FUNCTION_BLOCK "Asse_611U"	// FB 16
TITLE = Axis 611U management
AUTHOR : Cellini
VERSION : 0.1
VAR_INPUT
  IO_LAddr : INT ;	//Logic address of the inputs/outputs
END_VAR
VAR
  In_Profibus : STRUCT 	//Inputs from 611U (via Profibus)
   PKW : STRUCT 	//Parameter area of the Profibus telegram
    PKE : WORD ;
    IND : WORD ;
    PWE : DINT ;
   END_STRUCT ;
   PZD : STRUCT 	//Process data area of the Profibus telegram
    ZSW1 : STRUCT 	//Status word 1
     Bit8 : BOOL ;	//Following error (0=following error outside the window error)
     Bit9 : BOOL ;	//DP control requested (1=DP master is requested to accept control)
     Bit10 : BOOL ;	//Reference position reached (1=end of traversing block reached)
     Bit11 : BOOL ;	//Reference point set (1=axis is referenced)
     Bit12 : BOOL ;	//Setpoint acknowledge (1=the traversing task is processed)
     Bit13 : BOOL ;	//Drive stationery (1=drive is not in movement)
     Bit14 : BOOL ;	//External block change selected
     Bit15 : BOOL ;	//Request passive referencing
     Bit0 : BOOL ;	//Ready to switch-on (1=ready to power-up)
     Bit1 : BOOL ;	//Ready or no fault (1=drive ready or no fault present)
     Bit2 : BOOL ;	//Controller enable (1=speed controller active and setpoint can be accepted)
     Bit3 : BOOL ;	//Fault present (1=fault present)
     Bit4 : BOOL ;	//No OFF2 (1=OFF2 not present)
     Bit5 : BOOL ;	//No OFF3 (1=OFF3 not present)
     Bit6 : BOOL ;	//Switch-on inhibit (1=power-on inhibit)
     Bit7 : BOOL ;	//Alarm present (1=alarm present)
    END_STRUCT ;
    AktSatz : STRUCT 	//Actual block status word
     Bit8 : BOOL ;	//Reserved
     Bit9 : BOOL ;	//Reserved
     Bit10 : BOOL ;	//Reserved
     Bit11 : BOOL ;	//Reserved
     Bit12 : BOOL ;	//Reserved
     Bit13 : BOOL ;	//Reserved
     Bit14 : BOOL ;	//Reserved
     Bit15 : BOOL ;	//MDI Active
     Bit0 : BOOL ;	//Bit 0 block selected
     Bit1 : BOOL ;	//Bit 1 block selected
     Bit2 : BOOL ;	//Bit 2 block selected
     Bit3 : BOOL ;	//Bit 3 block selected
     Bit4 : BOOL ;	//Bit 4 block selected
     Bit5 : BOOL ;	//Bit 5 block selected
     Bit6 : BOOL ;	//Reserved
     Bit7 : BOOL ;	//Reserved
    END_STRUCT ;
    PosZsw : STRUCT 	//Position status word
     Bit8 : BOOL ;	//Cam switching signal 1
     Bit9 : BOOL ;	//Cam switching signal 2
     Bit10 : BOOL ;	//Direct output 1 via the traversing block
     Bit11 : BOOL ;	//Direct output 2 via the traversing block
     Bit12 : BOOL ;	//Fixed endstop reached
     Bit13 : BOOL ;	//Fixed endstop clamping torque reached
     Bit14 : BOOL ;	//Traverse to fixed endstop active
     Bit15 : BOOL ;	//Teach-In executed
     Bit0 : BOOL ;	//Tracking mode active (1=tracking mode active)
     Bit1 : BOOL ;	//Velocity limiting (1=velocity is limited)
     Bit2 : BOOL ;	//Setpoint stationary (1=axis stationary on the setpoint side)
     Bit3 : BOOL ;	//In synchronism (1=slave drive is synchronized with the master drive)
     Bit4 : BOOL ;	//Axis moves forwards
     Bit5 : BOOL ;	//Axis moves backwards
     Bit6 : BOOL ;	//Minus software limit switch actuated
     Bit7 : BOOL ;	//Plus software limit switch actuated
    END_STRUCT ;
    ZSW2 : STRUCT 	//Status word 2
     Bit8 : BOOL ;	//Suppress fault 608 active
     Bit9 : BOOL ;	//n.u. (used only in the n-set mode)
     Bit10 : BOOL ;	//n.u. (used only in the n-set mode)
     Bit11 : BOOL ;	//n.u. (used only in the n-set mode)
     Bit12 : BOOL ;	//Slave sign-of-life
     Bit13 : BOOL ;	//Slave sign-of-life
     Bit14 : BOOL ;	//Slave sign-of-life
     Bit15 : BOOL ;	//Slave sign-of-life
     Bit0 : BOOL ;	//Bit 0 parameter set
     Bit1 : BOOL ;	//Bit 1 parameter set
     Bit2 : BOOL ;	//Bit 2 parameter set
     Bit3 : BOOL ;	//First speed setpoint filter inactive
     Bit4 : BOOL ;	//Rump-function generator inactive
     Bit5 : BOOL ;	//Open holding brake
     Bit6 : BOOL ;	//Integrator inhibit
     Bit7 : BOOL ;	//Parking axis selected
    END_STRUCT ;
    XretrP : DINT ;	//Actual position value
    DIG_IN : STRUCT 	//Digital inputs status
     Bit8 : BOOL ;
     Bit9 : BOOL ;
     Bit10 : BOOL ;
     Bit11 : BOOL ;
     Bit12 : BOOL ;
     Bit13 : BOOL ;
     Bit14 : BOOL ;
     Bit15 : BOOL ;
     Bit0 : BOOL ;	//Axis on home cam
     Bit1 : BOOL ;	//Axis on minus extra-corse limit switch
     Bit2 : BOOL ;	//Axis on plus extra-corse limit switch
     Bit3 : BOOL ;
     Bit4 : BOOL ;
     Bit5 : BOOL ;
     Bit6 : BOOL ;
     Bit7 : BOOL ;
    END_STRUCT ;
   END_STRUCT ;
  END_STRUCT ;
  Out_Profibus : STRUCT 	//Outputs to 611U (via Profibus)
   PKW : STRUCT 	//Parameter area of the Profibus telegram
    PKE : WORD ;
    IND : WORD ;
    PWE : DINT ;
   END_STRUCT ;
   PZD : STRUCT 	//Process data area of the Profibus telegram
    STW1 : STRUCT 	//Control word 1
     Bit8 : BOOL ;	//JOG1 (1=the drive traverse with the speed in P0108)
     Bit9 : BOOL ;	//JOG2 (1=the drive traverse with the speed in P0109)
     Bit10 : BOOL ;	//Control requested (Should be set 1 when ZSW1.9=1)
     Bit11 : BOOL ;	//Stop referencing (1=start the referencing point approach)
     Bit12 : BOOL ;	//Opening the holding brake for test purposes
     Bit13 : BOOL ;	//External block change (With a edge the external block changing is initiated)
     Bit14 : BOOL ;	//Reserved
     Bit15 : BOOL ;	//Request passive referencing
     Bit0 : BOOL ;	//OFF1 (1=enable)
     Bit1 : BOOL ;	//OFF2 (1=enable)
     Bit2 : BOOL ;	//OFF3 (1=enable)
     Bit3 : BOOL ;	//Pulse inhibit (0=the motor stop for inertia)
     Bit4 : BOOL ;	//Reject travel task (0=stop the motor and delete the distance to go)
     Bit5 : BOOL ;	//Intermediate stop (0=stop the motor but the process is continued with 0/1 edge)
     Bit6 : BOOL ;	//Activate travel task (With a edge the traversing block selected is started)
     Bit7 : BOOL ;	//Reset the fault memory (1=Reset the fault memory)
    END_STRUCT ;
    SatzAnw : STRUCT 	//Block selection control word
     Bit8 : BOOL ;	//Reserved
     Bit9 : BOOL ;	//Reserved
     Bit10 : BOOL ;	//Reserved
     Bit11 : BOOL ;	//Reserved
     Bit12 : BOOL ;	//Reserved
     Bit13 : BOOL ;	//Reserved
     Bit14 : BOOL ;	//Reserved
     Bit15 : BOOL ;	//Activate MDI
     Bit0 : BOOL ;	//Bit 0 block selection
     Bit1 : BOOL ;	//Bit 1 block selection
     Bit2 : BOOL ;	//Bit 2 block selection
     Bit3 : BOOL ;	//Bit 3 block selection
     Bit4 : BOOL ;	//Bit 4 block selection
     Bit5 : BOOL ;	//Bit 5 block selection
     Bit6 : BOOL ;	//Reserved
     Bit7 : BOOL ;	//Reserved
    END_STRUCT ;
    PosStw : STRUCT 	//Position control word
     Bit8 : BOOL ;	//Reserved
     Bit9 : BOOL ;	//Reserved
     Bit10 : BOOL ;	//Reserved
     Bit11 : BOOL ;	//Reserved
     Bit12 : BOOL ;	//Reserved
     Bit13 : BOOL ;	//Reserved
     Bit14 : BOOL ;	//Reserved
     Bit15 : BOOL ;	//Reserved
     Bit0 : BOOL ;	//Tracking operation (1=select tracking operation)
     Bit1 : BOOL ;	//Set reference point (0/1 edge=P0160 is assigned as actual value)
     Bit2 : BOOL ;	//Reference cams (1=the axis is located at reference cam)
     Bit3 : BOOL ;	//Fixed endstop (1=fixed endstop reached)
     Bit4 : BOOL ;	//Activate the coupling (0/1 edge=activate coupling set via P0410)
     BIt5 : BOOL ;	//Incremental jogging (1=jog in velocity and increments)
     Bit6 : BOOL ;	//Activate Teach-In (0/1=Activate Teach-In; 1/0=Reset Teach-In)
     Bit7 : BOOL ;	//Invert the angular encoder input
    END_STRUCT ;
    STW2 : STRUCT 	//Control word 2
     Bit8 : BOOL ;	//Suppress fault 608
     Bit9 : BOOL ;	//n.u. (used only in the n-set mode)
     Bit10 : BOOL ;	//n.u. (used only in the n-set mode)
     Bit11 : BOOL ;	//n.u. (used only in the n-set mode)
     Bit12 : BOOL ;	//Master sign-of-life
     Bit13 : BOOL ;	//Master sign-of-life
     Bit14 : BOOL ;	//Master sign-of-life
     Bit15 : BOOL ;	//Master sign-of-life
     Bit0 : BOOL ;	//Bit 0 parameter set changeover
     Bit1 : BOOL ;	//Bit 1 parameter set changeover
     Bit2 : BOOL ;	//Bit 2 parameter set changeover
     Bit3 : BOOL ;	//First speed setpoint filter disabled
     Bit4 : BOOL ;	//Rump-function generator enabled
     Bit5 : BOOL ;	//Reserved
     Bit6 : BOOL ;	//Integrator inhibit
     Bit7 : BOOL ;	//Select parking axis
    END_STRUCT ;
    Over : INT ;	//Percentage value for the velocity override
   END_STRUCT ;
  END_STRUCT ;
  Enable : BOOL ;	//Enable the drive
  Reset_Alarms : BOOL ;	//Reset the alarms
  Reset_Axis : BOOL ;	//Stop all the movements
  Start_Inc : BOOL ;	//Start incremental movement
  Start_Abs : BOOL ;	//Start absolute movement
  Start_Rep : BOOL ;	//Start repositioning movement
  Start_Ref : BOOL ;	//Start referencing movement
  Stop : BOOL ;	//Intermediate stop movement
  Jog_Forward : BOOL ;	//Jog forward command
  Jog_Backward : BOOL ;	//Jog backward command
  STAT58 : BOOL ;	//Reserved
  STAT57 : BOOL ;	//Reserved
  STAT56 : BOOL ;	//Reserved
  STAT55 : BOOL ;	//Reserved
  STAT54 : BOOL ;	//Reserved
  STAT53 : BOOL ;	//Reserved
  Step1_Inc : BOOL ;	//Step 1 for incremental movement management
  Step2_Inc : BOOL ;	//Step 2 for incremental movement management
  Step1_Abs : BOOL ;	//Step 1 for absolute movement management
  Step2_Abs : BOOL ;	//Step 2 for absolute movement management
  STAT36 : BOOL ;	//Reserved
  STAT35 : BOOL ;	//Reserved
  STAT34 : BOOL ;	//Reserved
  STAT33 : BOOL ;	//Reserved
  InZeroPosition : BOOL ;	//Axis in "zero" position
  AxisStationery : BOOL ;	//Axis stationery
  DriveOK : BOOL ;	//Drive OK
  BrakeOpen : BOOL ;	//Open holding brake request
  AxisOnHWHomeCam : BOOL ;	//Axis on hardware home cam
  AxisOnHWSwitchN : BOOL ;	//Axis on minus hardware extra-corse limit switch
  AxisOnHWSwitchP : BOOL ;	//Axis on plus hardware extra-corse limit switch
  AxisOnSWSwitchN : BOOL ;	//Axis on minus software extra-corse limit switch
  AxisOnSWSwitchP : BOOL ;	//Axis on plus software extra-corse limit switch
  STAT69 : BOOL ;	//Reserved
  STAT67 : BOOL ;	//Reserved
  STAT66 : BOOL ;	//Reserved
  STAT65 : BOOL ;	//Reserved
  STAT64 : BOOL ;	//Reserved
  STAT63 : BOOL ;	//Reserved
  STAT70 : BOOL ;	//Reserved
  Aux1 : BOOL ;	//Auxiliary for edge management
  Aux2 : BOOL ;	//Auxiliary for edge management
  Aux3 : BOOL ;	//Auxiliary for edge management
  Aux4 : BOOL ;	//Auxiliary for edge management
  Aux5 : BOOL ;	//Auxiliary for edge management
  Aux6 : BOOL ;	//Auxiliary for edge management
  Aux7 : BOOL ;	//Auxiliary for edge management
  Aux8 : BOOL ;	//Auxiliary for edge management
  Target_Inc : DINT ;	//Target for the incremental movement
  Target_Abs : DINT ;	//Target for the absolute movement
  DistanceToGo_Abs : DINT ;	//Difference between actual and new position
  Override : INT ;	//Percentage value for the velocity override
  ActualPosition : DINT ;	//Actual position value
END_VAR
VAR_TEMP
  tempAR1 : DWORD ;
  tempAR2 : DWORD ;
  tempSRC : ANY ;
  tempDST : ANY ;
  tempDWORD_1 : DWORD ;
  tempWORD_1 : WORD ;
  tempINT : INT ;
  tempDWORD_2 : DWORD ;
END_VAR
BEGIN
NETWORK
TITLE = Mapping of the inputs
      L     #IO_LAddr;
      SLD   3;
      T     #tempDWORD_1;
      L     P##In_Profibus;
      T     #tempDWORD_2;
      L     11;
NXT1: T     #tempINT;
      L     PIW [#tempDWORD_1];
      T     DIW [#tempDWORD_2];
      L     #tempDWORD_1;
      L     P#2.0;
      +D;
      T     #tempDWORD_1;
      L     #tempDWORD_2;
      L     P#2.0;
      +D;
      T     #tempDWORD_2;
      L     #tempINT;
      LOOP  NXT1;
NETWORK
TITLE = Status
//Axis stationery
      A     #In_Profibus.PZD.ZSW1.Bit13;
      AN    #In_Profibus.PZD.ZSW1.Bit12;
      =     #AxisStationery;
//Drive OK
      A     #In_Profibus.PZD.ZSW1.Bit0;
      A     #In_Profibus.PZD.ZSW1.Bit1;
      A     #In_Profibus.PZD.ZSW1.Bit2;
      AN    #In_Profibus.PZD.ZSW1.Bit3;
      A     #In_Profibus.PZD.ZSW1.Bit4;
      A     #In_Profibus.PZD.ZSW1.Bit5;
      A     #In_Profibus.PZD.ZSW1.Bit8;
      =     #DriveOK;
//Open holding brake request
      A     #In_Profibus.PZD.ZSW2.Bit5;
      =     #BrakeOpen;
//Axis on hardware home cam
      A     #In_Profibus.PZD.DIG_IN.Bit0;
      =     #AxisOnHWHomeCam;
//Axis on hardware minus extra-course limit switch
      A     #In_Profibus.PZD.DIG_IN.Bit1;
      =     #AxisOnHWSwitchN;
//Axis on hardware plus extra-course limit switch
      A     #In_Profibus.PZD.DIG_IN.Bit2;
      =     #AxisOnHWSwitchP;
//Axis on software minus extra-course limit switch
      A     #In_Profibus.PZD.PosZsw.Bit6;
      =     #AxisOnSWSwitchN;
//Axis on software plus extra-course limit switch
      A     #In_Profibus.PZD.PosZsw.Bit7;
      =     #AxisOnSWSwitchP;
//Actual position value
      L     #In_Profibus.PZD.XretrP;
      T     #ActualPosition;
NETWORK
TITLE = Commands
//Enable the drive
      A     #Enable;
      =     #Out_Profibus.PZD.STW1.Bit0;
      =     #Out_Profibus.PZD.STW1.Bit1;
      =     #Out_Profibus.PZD.STW1.Bit2;
      A     "On";
      =     #Out_Profibus.PZD.STW1.Bit3;
//Erase all the movements
      O     #Reset_Axis;
      O     #In_Profibus.PZD.ZSW1.Bit3;
      ON    #In_Profibus.PZD.ZSW1.Bit8;
      R     #Start_Inc;
      R     #Step1_Inc;
      R     #Step2_Inc;
      R     #Start_Abs;
      R     #Step1_Abs;
      R     #Step2_Abs;
      R     #Start_Rep;
      R     #Start_Ref;
      R     #Out_Profibus.PZD.STW1.Bit11;
      R     #Out_Profibus.PZD.STW1.Bit6;
//Stop the axis and erase the distance to go
      AN    #Reset_Axis;
      =     #Out_Profibus.PZD.STW1.Bit4;
//Intermediate stop the axis (the movement continued with a 0/1 edge)
      AN    #Stop;
      =     #Out_Profibus.PZD.STW1.Bit5;
//Reset alarms
      A     #Reset_Alarms;
      =     #Out_Profibus.PZD.STW1.Bit7;
//Control request (611U<->PLC communication)
      A     #In_Profibus.PZD.ZSW1.Bit9;
      =     #Out_Profibus.PZD.STW1.Bit10;
//Velocity override
      L     #Override;
      T     #Out_Profibus.PZD.Over;
NETWORK
TITLE = Movement in incremental mode
//Reset the incremental movement if the axis is the distance to go is minus then 0,05mm
      A     #Start_Inc;
      A(;
      L     #Target_Inc;
      L     50;
      <D;
      );
      A(;
      L     #Target_Inc;
      L     -50;
      >D;
      );
      R     #Start_Inc;
//Select the travel block (Block number 2=000010)
      A     #Start_Inc;
      R     #Out_Profibus.PZD.SatzAnw.Bit0;
      S     #Out_Profibus.PZD.SatzAnw.Bit1;
      R     #Out_Profibus.PZD.SatzAnw.Bit2;
      R     #Out_Profibus.PZD.SatzAnw.Bit3;
      R     #Out_Profibus.PZD.SatzAnw.Bit4;
      R     #Out_Profibus.PZD.SatzAnw.Bit5;
//Load the new position of the travel block
      A     #Start_Inc;
      AN    #Step1_Inc;
      AN    #Step2_Inc;
      S     #Step1_Inc;
      JCN   L001;
      L     #Target_Inc;
      T     #Out_Profibus.PKW.PWE;
      L     W#16#8051;
      T     #Out_Profibus.PKW.PKE;
      L     2;
      T     #Out_Profibus.PKW.IND;
L001: NOP   0;
//Check if the 611U received the change
      A     #Start_Inc;
      A     #Step1_Inc;
      AN    #Step2_Inc;
      A(;
      L     #Out_Profibus.PKW.PWE;
      L     #In_Profibus.PKW.PWE;
      ==D;
      );
      A(;
      L     W#16#5051;
      L     #In_Profibus.PKW.PKE;
      ==I;
      );
      A(;
      L     #Out_Profibus.PKW.IND;
      L     #In_Profibus.PKW.IND;
      ==I;
      );
      S     #Step2_Inc;
//Start travel task
      A     #Start_Inc;
      A     #Step1_Inc;
      A     #Step2_Inc;
      A(;
      L     #Target_Inc;
      L     #In_Profibus.PKW.PWE;
      ==D;
      );
//UN    #In_Profibus.PZD.AktSatz.Bit0
//U     #In_Profibus.PZD.AktSatz.Bit1
//UN    #In_Profibus.PZD.AktSatz.Bit2
//UN    #In_Profibus.PZD.AktSatz.Bit3
//UN    #In_Profibus.PZD.AktSatz.Bit4
//UN    #In_Profibus.PZD.AktSatz.Bit5
      AN    #Out_Profibus.PZD.STW1.Bit6;
      S     #Out_Profibus.PZD.STW1.Bit6;
      JCN   L002;
      L     0;
      T     #Out_Profibus.PKW.PKE;
      T     #Out_Profibus.PKW.IND;
      T     #Out_Profibus.PKW.PWE;
L002: NOP   0;
//End incremental movement
      A     #In_Profibus.PZD.ZSW1.Bit10;
      FP    #Aux1;
      A     #Start_Inc;
      A     #Step1_Inc;
      A     #Step2_Inc;
      A     #Out_Profibus.PZD.STW1.Bit6;
      R     #Out_Profibus.PZD.STW1.Bit6;
      R     #Start_Inc;
      R     #Step1_Inc;
      R     #Step2_Inc;
NETWORK
TITLE = Movement in absolute mode
//Movement not necessary if the axis is just in position  
      A     #Start_Abs;
      AN    #Step1_Abs;
      AN    #Step2_Abs;
      JCN   L004;
//Calculate the difference between the actual position and new position
      L     #Target_Abs;
      L     #In_Profibus.PZD.XretrP;
      -D;
      T     #DistanceToGo_Abs;
      L     0;
      <D;
      JCN   L003;
      L     #DistanceToGo_Abs;
      NEGD;
      T     #DistanceToGo_Abs;
L003: NOP   0;
      A(;
      L     #DistanceToGo_Abs;
      L     99;
      <=D;
      );
      R     #Start_Abs;
L004: NOP   0;
//Select the travel block (Block number 0=000000)
      A     #Start_Abs;
      R     #Out_Profibus.PZD.SatzAnw.Bit0;
      R     #Out_Profibus.PZD.SatzAnw.Bit1;
      R     #Out_Profibus.PZD.SatzAnw.Bit2;
      R     #Out_Profibus.PZD.SatzAnw.Bit3;
      R     #Out_Profibus.PZD.SatzAnw.Bit4;
      R     #Out_Profibus.PZD.SatzAnw.Bit5;
//Load the new position of the travel block
      A     #Start_Abs;
      AN    #Step1_Abs;
      AN    #Step2_Abs;
      S     #Step1_Abs;
      JCN   L005;
      L     #Target_Abs;
      T     #Out_Profibus.PKW.PWE;
      L     W#16#8051;
      T     #Out_Profibus.PKW.PKE;
      L     0;
      T     #Out_Profibus.PKW.IND;
L005: NOP   0;
//Check if the 611U received the change
      A     #Start_Abs;
      A     #Step1_Abs;
      AN    #Step2_Abs;
      A(;
      L     #Out_Profibus.PKW.PWE;
      L     #In_Profibus.PKW.PWE;
      ==D;
      );
      A(;
      L     W#16#5051;
      L     #In_Profibus.PKW.PKE;
      ==I;
      );
      A(;
      L     #Out_Profibus.PKW.IND;
      L     #In_Profibus.PKW.IND;
      ==I;
      );
      S     #Step2_Abs;
//Start travel task
      A     #Start_Abs;
      A     #Step1_Abs;
      A     #Step2_Abs;
      A(;
      L     #Target_Abs;
      L     #In_Profibus.PKW.PWE;
      ==D;
      );
      AN    #In_Profibus.PZD.AktSatz.Bit0;
      AN    #In_Profibus.PZD.AktSatz.Bit1;
      AN    #In_Profibus.PZD.AktSatz.Bit2;
      AN    #In_Profibus.PZD.AktSatz.Bit3;
      AN    #In_Profibus.PZD.AktSatz.Bit4;
      AN    #In_Profibus.PZD.AktSatz.Bit5;
      AN    #Out_Profibus.PZD.STW1.Bit6;
      S     #Out_Profibus.PZD.STW1.Bit6;
      JCN   L006;
      L     0;
      T     #Out_Profibus.PKW.PKE;
      T     #Out_Profibus.PKW.IND;
      T     #Out_Profibus.PKW.PWE;
L006: NOP   0;
//End absolute movement
      A     #In_Profibus.PZD.ZSW1.Bit10;
      FP    #Aux2;
      A     #Start_Abs;
      A     #Step1_Abs;
      A     #Step2_Abs;
      A     #Out_Profibus.PZD.STW1.Bit6;
      R     #Out_Profibus.PZD.STW1.Bit6;
      R     #Start_Abs;
      R     #Step1_Abs;
      R     #Step2_Abs;
NETWORK
TITLE = Repositioning management
//Movement not necessary if the axis is just in position  
      A     #Start_Rep;
      FP    #Aux3;
      A     #InZeroPosition;
      R     #Start_Rep;
//Select the travel block (Block number 1=000001)
      A     #Start_Rep;
      S     #Out_Profibus.PZD.SatzAnw.Bit0;
      R     #Out_Profibus.PZD.SatzAnw.Bit1;
      R     #Out_Profibus.PZD.SatzAnw.Bit2;
      R     #Out_Profibus.PZD.SatzAnw.Bit3;
      R     #Out_Profibus.PZD.SatzAnw.Bit4;
      R     #Out_Profibus.PZD.SatzAnw.Bit5;
//Start travel task
      A     #Start_Rep;
      A     #In_Profibus.PZD.AktSatz.Bit0;
      AN    #In_Profibus.PZD.AktSatz.Bit1;
      AN    #In_Profibus.PZD.AktSatz.Bit2;
      AN    #In_Profibus.PZD.AktSatz.Bit3;
      AN    #In_Profibus.PZD.AktSatz.Bit4;
      AN    #In_Profibus.PZD.AktSatz.Bit5;
      AN    #Out_Profibus.PZD.STW1.Bit6;
      S     #Out_Profibus.PZD.STW1.Bit6;
//End repositioning
      A     #In_Profibus.PZD.ZSW1.Bit10;
      FP    #Aux4;
      A     #Start_Rep;
      A     #Out_Profibus.PZD.STW1.Bit6;
      R     #Out_Profibus.PZD.STW1.Bit6;
      R     #Start_Rep;
NETWORK
TITLE = Jog management
//Jog forward
      A     #Jog_Forward;
      A     #In_Profibus.PZD.ZSW1.Bit11;
      AN    #In_Profibus.PZD.PosZsw.Bit7;
      =     #Out_Profibus.PZD.STW1.Bit9;
//Jog backward
      A     #Jog_Backward;
      A     #In_Profibus.PZD.ZSW1.Bit11;
      AN    #In_Profibus.PZD.PosZsw.Bit6;
      =     #Out_Profibus.PZD.STW1.Bit8;
NETWORK
TITLE = Referencing management
//Start the referencing point approach
      A     #Start_Ref;
      FP    #Aux5;
      S     #Out_Profibus.PZD.STW1.Bit11;
//End of referencing point approch
      A     #In_Profibus.PZD.ZSW1.Bit11;
      FP    #Aux6;
      R     #Out_Profibus.PZD.STW1.Bit11;
      R     #Start_Ref;
NETWORK
TITLE = Mapping of the outputs
      L     #IO_LAddr;
      SLD   3;
      T     #tempDWORD_1;
      L     P##Out_Profibus;
      T     #tempDWORD_2;
      L     9;
NXT3: T     #tempINT;
      L     DIW [#tempDWORD_2];
      T     PQW [#tempDWORD_1];
      L     #tempDWORD_1;
      L     P#2.0;
      +D;
      T     #tempDWORD_1;
      L     #tempDWORD_2;
      L     P#2.0;
      +D;
      T     #tempDWORD_2;
      L     #tempINT;
      LOOP  NXT3;
END_FUNCTION_BLOCK

FUNCTION_BLOCK "BALLUFF"	// FB 20
TITLE = BALLUFF Reader/Writer management
AUTHOR : Salvati
VERSION : 0.1
VAR_INPUT
  IO_LAddr : INT ;
END_VAR
VAR
  InputBuffer : STRUCT
   CP : BOOL ;	//Codetag present
   AA : BOOL ;	//Command started
   AE : BOOL ;	//Command finished without error
   AF : BOOL ;	//Command finished with error
   KN : BOOL ;	//Header number
   TO : BOOL ;	//Toggle-bit Out
   HF : BOOL ;	//Head error
   BB : BOOL ;	//Ready
   ErrorCode : BYTE ;
   Data1 : BYTE ;
   Data2 : BYTE ;
   Data3 : BYTE ;
   Data4 : BYTE ;
  END_STRUCT ;
  OutputBuffer : STRUCT
   AV : BOOL ;	//Command
   Reserved1 : BOOL ;
   GR : BOOL ;	//Ground state
   Reserved2 : BOOL ;
   HD : BOOL ;	//Head direct
   Reserved3 : BOOL ;
   TI : BOOL ;	//Toggle-bit in
   CT : BOOL ;	//Codetag type
   Command : BYTE ;
   StartAddress_L : BYTE ;
   StartAddress_H : BYTE ;
   NoBytes_L : BYTE ;
   NoBytes_H : BYTE ;
  END_STRUCT ;
  Testa1 : STRUCT
   Lettura_Start : BOOL ;	//1=start read job
   Lettura_OK : BOOL ;	//1=read job ended without error
   Lettura_NOK : BOOL ;	//1=read job ended with error
   Lettura_Step1 : BOOL ;	//Aux for read job cycle
   Lettura_Step2 : BOOL ;	//Aux for read job cycle
   Lettura_Step3 : BOOL ;	//Aux for read job cycle
   Lettura_Step4 : BOOL ;	//Aux for read job cycle
   Lettura_Step5 : BOOL ;	//Aux for read job cycle
   Scrittura_Start : BOOL ;	//1=start write job
   Scrittura_OK : BOOL ;	//1=write job ended without error
   Scrittura_NOK : BOOL ;	//1=write job ended with error
   Scrittura_Step1 : BOOL ;	//Aux for write job cycle
   Scrittura_Step2 : BOOL ;	//Aux for write job cycle
   Scrittura_Step3 : BOOL ;	//Aux for write job cycle
   Scrittura_Step4 : BOOL ;	//Aux for write job cycle
   Scrittura_Step5 : BOOL ;	//Aux for write job cycle
   ValoreLetto : BYTE ;	//Data readed
   ValoreDaScrivere : BYTE ;	//Data to write
   Seconds : BYTE ;	//Number of seconds of activity
  END_STRUCT ;
  Testa2 : STRUCT
   Lettura_Start : BOOL ;	//1=start read job
   Lettura_OK : BOOL ;	//1=read job ended without error
   Lettura_NOK : BOOL ;	//1=read job ended with error
   Lettura_Step1 : BOOL ;	//Aux for read job cycle
   Lettura_Step2 : BOOL ;	//Aux for read job cycle
   Lettura_Step3 : BOOL ;	//Aux for read job cycle
   Lettura_Step4 : BOOL ;	//Aux for read job cycle
   Lettura_Step5 : BOOL ;	//Aux for read job cycle
   Scrittura_Start : BOOL ;	//1=start write job
   Scrittura_OK : BOOL ;	//1=write job ended without error
   Scrittura_NOK : BOOL ;	//1=write job ended with error
   Scrittura_Step1 : BOOL ;	//Aux for write job cycle
   Scrittura_Step2 : BOOL ;	//Aux for write job cycle
   Scrittura_Step3 : BOOL ;	//Aux for write job cycle
   Scrittura_Step4 : BOOL ;	//Aux for write job cycle
   Scrittura_Step5 : BOOL ;	//Aux for write job cycle
   ValoreLetto : BYTE ;	//Data readed
   ValoreDaScrivere : BYTE ;	//Data to write
   Seconds : BYTE ;	//Number of seconds of activity
  END_STRUCT ;
END_VAR
VAR_TEMP
  tempAR1 : DWORD ;
  tempAR2 : DWORD ;
  tempSRC : ANY ;
  tempDST : ANY ;
  tempDWORD_1 : DWORD ;
  tempWORD_1 : WORD ;
  tempINT : INT ;
  tempBYTE1 : BYTE ;
  tempBYTE2 : BYTE ;
END_VAR
BEGIN
NETWORK
TITLE = Mapping of the inputs
//Save registry value
      TAR1  #tempAR1;
      TAR2  #tempAR2;
//Creation of a pointer to the source area
      LAR1  P##tempSRC;	//Load initial address of source pointer in AR1
      L     B#16#10;	//Load the ID for the ANY type
      T     LB [AR1,P#0.0];
      L     B#16#2;	//2=type of data is BYTE
      T     LB [AR1,P#1.0];
      L     6;	//Number of bytess to transfer
      T     LW [AR1,P#2.0];
      L     0;	//Type of data memory
      T     LW [AR1,P#4.0];
      L     DIW 0;
      SLD   3;
      L     P#I 0.0;
      +D;
      T     LD [AR1,P#6.0];
//Creation of a pointer to the target area
      LAR1  P##tempDST;	//Load initial address of destination pointer in AR1
      L     B#16#10;	//Load the ID for the ANY type
      T     LB [AR1,P#0.0];
      L     B#16#2;	//2=type of data is BYTE
      T     LB [AR1,P#1.0];
      L     6;	//Number of bytes to receive
      T     LW [AR1,P#2.0];
      L     0;	//Type of data memory
      T     LW [AR1,P#4.0];
      L     P##InputBuffer;
      T     LD [AR1,P#6.0];
//Trasfering data
      CALL  "BLKMOV" (
           SRCBLK                   := #tempSRC,
           RET_VAL                  := #tempINT,
           DSTBLK                   := #tempDST);
//Load saved registry value
      LAR1  #tempAR1;
      LAR2  #tempAR2;
NETWORK
TITLE = Mapping of the outputs
//Save registry value
      TAR1  #tempAR1;
      TAR2  #tempAR2;
//Creation of a pointer to the source area
      LAR1  P##tempSRC;	//Load initial address of source pointer in AR1
      L     B#16#10;	//Load the ID for the ANY type
      T     LB [AR1,P#0.0];
      L     B#16#2;	//2=type of data is BYTE
      T     LB [AR1,P#1.0];
      L     6;	//Number of bytess to transfer
      T     LW [AR1,P#2.0];
      L     0;	//Type of data memory
      T     LW [AR1,P#4.0];
      L     DIW 0;
      SLD   3;
      L     P#Q 0.0;
      +D;
      T     LD [AR1,P#6.0];
//Creation of a pointer to the target area
      LAR1  P##tempDST;	//Load initial address of destination pointer in AR1
      L     B#16#10;	//Load the ID for the ANY type
      T     LB [AR1,P#0.0];
      L     B#16#2;	//2=type of data is BYTE
      T     LB [AR1,P#1.0];
      L     6;	//Number of bytes to receive
      T     LW [AR1,P#2.0];
      L     0;	//Type of data memory
      T     LW [AR1,P#4.0];
      L     P##OutputBuffer;
      T     LD [AR1,P#6.0];
//Trasfering data
      CALL  "BLKMOV" (
           SRCBLK                   := #tempSRC,
           RET_VAL                  := #tempINT,
           DSTBLK                   := #tempDST);
//Load saved registry value
      LAR1  #tempAR1;
      LAR2  #tempAR2;
NETWORK
TITLE = Read job of header 1
      A     DIX 14.3;
      A     "Clock_P";
      JCN   L006;
      L     DIB 18;
      L     1;
      +I;
      T     DIB 18;
L006: NOP   0;
//Select the header
      A     DIX 14.0;
      AN    DIX 15.0;
//UN    #Testa2.Lettura_Start
//UN    #Testa2.Scrittura_Start
      AN    DIX 14.3;
      S     DIX 14.3;
      R     DIX 8.4;
      JCN   L005;
      L     0;
      T     DIB 18;
L005: NOP   0;
//Check the header selected
      A     DIX 14.0;
      A     DIX 14.3;
      AN    DIX 2.4;
      AN    DIX 14.4;
      S     DIX 14.4;
//Start reading job
      A     DIX 14.0;
      A     DIX 14.4;
      A     DIX 2.7;
      A     DIX 2.0;
      AN    DIX 14.5;
      S     DIX 14.5;
      R     DIX 14.1;
      R     DIX 14.2;
      S     DIX 8.0;
      R     DIX 8.7;
      JC    L001;
      JU    L004;
L001: NOP   0;
      L     0;
      T     DIB 10;
      T     DIB 11;
      T     DIB 13;
      L     1;
      T     DIB 12;
      L     1;
      T     DIB 9;
L004: NOP   0;
//Read job ended with error
      A     DIX 14.0;
      A     DIX 14.5;
      A     DIX 2.1;
      A     DIX 2.3;
      O;
      A(;
      L     DIB 18;
      L     10;
      >=I;
      );
      R     DIX 14.3;
      R     DIX 14.4;
      R     DIX 14.5;
      R     DIX 8.0;
      R     DIX 14.0;
      S     DIX 14.2;
      JCN   L007;
      L     0;
      T     DIB 18;
L007: NOP   0;
//Read job ended without error
      A     DIX 14.0;
      A     DIX 14.5;
      A     DIX 2.1;
      A     DIX 2.2;
      R     DIX 14.3;
      R     DIX 14.4;
      R     DIX 14.5;
      R     DIX 8.0;
      R     DIX 14.0;
      S     DIX 14.1;
      JC    L002;
      JU    L003;
L002: L     DIB 3;
//T     #tempBYTE1
//L     #InputBuffer.Data1
//T     #tempBYTE2
//L     LW    36
      T     DIB 16;
L003: NOP   0;
NETWORK
TITLE = Write job of header 1
      A     DIX 15.3;
      A     "Clock_P";
      JCN   L018;
      L     DIB 18;
      L     1;
      +I;
      T     DIB 18;
L018: NOP   0;
//Select the header
      A     DIX 15.0;
      AN    DIX 14.0;
//UN    #Testa2.Lettura_Start
//UN    #Testa2.Scrittura_Start
      AN    DIX 15.3;
      S     DIX 15.3;
      R     DIX 8.4;
      JCN   L015;
      L     0;
      T     DIB 18;
L015: NOP   0;
//Check the header selected
      A     DIX 15.0;
      A     DIX 15.3;
      AN    DIX 2.4;
      AN    DIX 15.4;
      S     DIX 15.4;
//Start writing job
      A     DIX 15.0;
      A     DIX 15.4;
      A     DIX 2.7;
      A     DIX 2.0;
      AN    DIX 15.5;
      S     DIX 15.5;
      R     DIX 15.1;
      R     DIX 15.2;
      S     DIX 8.0;
      R     DIX 8.7;
      JC    L011;
      JU    L012;
L011: NOP   0;
      L     0;
      T     DIB 10;
      T     DIB 11;
      T     DIB 13;
      L     1;
      T     DIB 12;
      L     2;
      T     DIB 9;
L012: NOP   0;
//Confirm write job in course
      A     DIX 15.0;
      A     DIX 15.5;
      A     DIX 2.1;
      A     DIX 2.5;
      AN    DIX 15.6;
      S     DIX 15.6;
      S     DIX 8.6;
      JC    L016;
      JU    L017;
L016: NOP   0;
      L     DIB 17;
//T     LW    36
//L     #tempBYTE1
      T     DIB 9;
//L     #tempBYTE2
//T     #OutputBuffer.StartAddress_L
L017: NOP   0;
//Write job ended with error
      A     DIX 15.0;
      A     DIX 15.6;
      A     DIX 2.1;
      A     DIX 2.3;
      O;
      A(;
      L     DIB 18;
      L     10;
      >=I;
      );
      R     DIX 15.3;
      R     DIX 15.4;
      R     DIX 15.5;
      R     DIX 15.6;
      R     DIX 8.0;
      R     DIX 8.6;
      R     DIX 15.0;
      S     DIX 15.2;
      JCN   L019;
      L     0;
      T     DIB 18;
L019: NOP   0;
//Write job ended without error
      A     DIX 15.0;
      A     DIX 15.6;
      A     DIX 2.1;
      A     DIX 2.2;
      R     DIX 15.3;
      R     DIX 15.4;
      R     DIX 15.5;
      R     DIX 15.6;
      R     DIX 8.0;
      R     DIX 8.6;
      R     DIX 15.0;
      S     DIX 15.1;
NETWORK
TITLE = Read job of header 2
      A     DIX 20.3;
      A     "Clock_P";
      JCN   L026;
      L     DIB 24;
      L     1;
      +I;
      T     DIB 24;
L026: NOP   0;
//Select the header
      A     DIX 20.0;
      AN    DIX 21.0;
      AN    DIX 14.0;
      AN    DIX 15.0;
      AN    DIX 20.3;
      S     DIX 20.3;
      S     DIX 8.4;
      JCN   L025;
      L     0;
      T     DIB 24;
L025: NOP   0;
//Check the header selected
      A     DIX 20.0;
      A     DIX 20.3;
      A     DIX 2.4;
      AN    DIX 20.4;
      S     DIX 20.4;
//Start reading job
      A     DIX 20.0;
      A     DIX 20.4;
      A     DIX 2.7;
      A     DIX 2.0;
      AN    DIX 20.5;
      S     DIX 20.5;
      R     DIX 20.1;
      R     DIX 20.2;
      S     DIX 8.0;
      R     DIX 8.7;
      JC    L021;
      JU    L024;
L021: NOP   0;
      L     0;
      T     DIB 10;
      T     DIB 11;
      T     DIB 13;
      L     1;
      T     DIB 12;
      L     1;
      T     DIB 9;
L024: NOP   0;
//Read job ended with error
      A     DIX 20.0;
      A     DIX 20.5;
      A     DIX 2.1;
      A     DIX 2.3;
      O;
      A(;
      L     DIB 24;
      L     10;
      >=I;
      );
      R     DIX 20.3;
      R     DIX 20.4;
      R     DIX 20.5;
      R     DIX 8.0;
      R     DIX 20.0;
      S     DIX 20.2;
      JCN   L027;
      L     0;
      T     DIB 24;
L027: NOP   0;
//Read job ended without error
      A     DIX 20.0;
      A     DIX 20.5;
      A     DIX 2.1;
      A     DIX 2.2;
      R     DIX 20.3;
      R     DIX 20.4;
      R     DIX 20.5;
      R     DIX 8.0;
      R     DIX 20.0;
      S     DIX 20.1;
      JC    L022;
      JU    L023;
L022: L     DIB 3;
//T     #tempBYTE1
//L     #InputBuffer.Data1
//T     #tempBYTE2
//L     LW    36
      T     DIB 22;
L023: NOP   0;
NETWORK
TITLE = Write job of header 2
      A     DIX 21.3;
      A     "Clock_P";
      JCN   L038;
      L     DIB 24;
      L     1;
      +I;
      T     DIB 24;
L038: NOP   0;
//Select the header
      A     DIX 21.0;
      AN    DIX 20.0;
      AN    DIX 14.0;
      AN    DIX 15.0;
      AN    DIX 21.3;
      S     DIX 21.3;
      S     DIX 8.4;
      JCN   L035;
      L     0;
      T     DIB 24;
L035: NOP   0;
//Check the header selected
      A     DIX 21.0;
      A     DIX 21.3;
      A     DIX 2.4;
      AN    DIX 21.4;
      S     DIX 21.4;
//Start writing job
      A     DIX 21.0;
      A     DIX 21.4;
      A     DIX 2.7;
      A     DIX 2.0;
      AN    DIX 21.5;
      S     DIX 21.5;
      R     DIX 21.1;
      R     DIX 21.2;
      S     DIX 8.0;
      R     DIX 8.7;
      JC    L031;
      JU    L032;
L031: NOP   0;
      L     0;
      T     DIB 10;
      T     DIB 11;
      T     DIB 13;
      L     1;
      T     DIB 12;
      L     2;
      T     DIB 9;
L032: NOP   0;
//Confirm write job in course
      A     DIX 21.0;
      A     DIX 21.5;
      A     DIX 2.1;
      A     DIX 2.5;
      AN    DIX 21.6;
      S     DIX 21.6;
      S     DIX 8.6;
      JC    L036;
      JU    L037;
L036: NOP   0;
      L     DIB 23;
//T     LW    36
//L     #tempBYTE1
      T     DIB 9;
//L     #tempBYTE2
//T     #OutputBuffer.StartAddress_L
L037: NOP   0;
//Write job ended with error
      A     DIX 21.0;
      A     DIX 21.6;
      A     DIX 2.1;
      A     DIX 2.3;
      O;
      A(;
      L     DIB 24;
      L     10;
      >=I;
      );
      R     DIX 21.3;
      R     DIX 21.4;
      R     DIX 21.5;
      R     DIX 21.6;
      R     DIX 8.0;
      R     DIX 8.6;
      R     DIX 21.0;
      S     DIX 21.2;
      JCN   L039;
      L     0;
      T     DIB 24;
L039: NOP   0;
//Write job ended without error
      A     DIX 21.0;
      A     DIX 21.6;
      A     DIX 2.1;
      A     DIX 2.2;
      R     DIX 21.3;
      R     DIX 21.4;
      R     DIX 21.5;
      R     DIX 21.6;
      R     DIX 8.0;
      R     DIX 8.6;
      R     DIX 21.0;
      S     DIX 21.1;
NETWORK
TITLE = Mapping of the outputs
//Save registry value
      TAR1  #tempAR1;
      TAR2  #tempAR2;
//Creation of a pointer to the source area
      LAR1  P##tempSRC;	//Load initial address of source pointer in AR1
      L     B#16#10;	//Load the ID for the ANY type
      T     LB [AR1,P#0.0];
      L     B#16#2;	//2=type of data is BYTE
      T     LB [AR1,P#1.0];
      L     6;	//Number of bytess to transfer
      T     LW [AR1,P#2.0];
      L     0;	//Type of data memory
      T     LW [AR1,P#4.0];
      L     P##OutputBuffer;
      T     LD [AR1,P#6.0];
//Creation of a pointer to the target area
      LAR1  P##tempDST;	//Load initial address of destination pointer in AR1
      L     B#16#10;	//Load the ID for the ANY type
      T     LB [AR1,P#0.0];
      L     B#16#2;	//2=type of data is BYTE
      T     LB [AR1,P#1.0];
      L     6;	//Number of bytes to receive
      T     LW [AR1,P#2.0];
      L     0;	//Type of data memory
      T     LW [AR1,P#4.0];
      L     DIW 0;
      SLD   3;
      L     P#Q 0.0;
      +D;
      T     LD [AR1,P#6.0];
//Trasfering data
      CALL  "BLKMOV" (
           SRCBLK                   := #tempSRC,
           RET_VAL                  := #tempINT,
           DSTBLK                   := #tempDST);
//Load saved registry value
      LAR1  #tempAR1;
      LAR2  #tempAR2;
END_FUNCTION_BLOCK

FUNCTION_BLOCK "FB24 - Gestione Mov Assi"	// FB 24
TITLE = GESTIONE ASSI STAZIONE OP60
VERSION : 0.1
VAR_INPUT
  INDIRIZZO_INIZIALE_E_A : DINT ;	//INDIRIZZO INIZIALE I/O (VEDI CONFIGURAZIONE HARDWARE)
  OK_FOR_COMMANDS : BOOL ;	//TUTTO PRONTO PER I COMANDI
  RESET_ALLARMI : BOOL ;	//1=RESET ALLARMI AZIONAMENTO
  STOP : BOOL ;	//0=STOP DI TUTTI I MOVIMENTI
  TARGET_POSIZIONE : DINT ;	//TARGET DI POSIZIONAMENTO ASSOLUTO
  TARGET_INCREMENTALE : DINT ;	//SPOSTAMENTO IN MODO INCREMENTALE
  OVERRIDE : INT ;	//OVVERIDE DI VELOCITA'
  JOG_PIU : BOOL ;	//COMANDO JOG PIU'
  JOG_MENO : BOOL ;	//COMANDO JOG MENO
  IN_PKE : WORD ;
  IN_IND : WORD ;
  IN_PWE : DINT ;
  ASSE_SU_HOME : BOOL ;	//ASSE GIA' SU POSIZIONE DI HOME
END_VAR
VAR_OUTPUT
  OUT_PKE : WORD ;
  OUT_IND : WORD ;
  OUT_PWE : DINT ;
  POSIZIONE_ATTUALE : DINT ;
  POSIZIONE_RAGGIUNTA : BOOL ;	//POSIZIONAMENTO ULTIMATO
  HOME_OK : BOOL ;	//1=ASSE RIFERITO
  RIPOSIZIONAMENTO_OK : BOOL ;	//1=RIPOSIZIONAMENTO EFFETTUATO
  ASSE_FERMO_NO_JOB : BOOL ;	//1=ASSE FERMO E NESSUN JOB IN CORSO
  AZIONAMENTO_OK : BOOL ;	//1=AZIONAMENTO PRONTO
  AZIONAMENTO_FAULT : BOOL ;	//1=AZIONAMENTO IN ALLARME
  CAMMA_DI_RIFERIMENTO : BOOL ;	//1=ASSE SU CAMMA DI RIFERIMENTO
  OLTRECORSA_NEGATIVO : BOOL ;	//1=ASSE SU OLTRECORSA HARDWARE NEGATIVO
  OLTRECORSA_POSITIVO : BOOL ;	//1=ASSE SU OLTRECORSA HARDWARE POSITIVO
  FINECORSA_SOFTWARE_NEG : BOOL ;	//1=FINECORSA SOFTWARE NEGATIVO
  FINECORSA_SOFTWARE_POS : BOOL ;	//1=FINECORSA SOFTWARE POSITIVO
  FRENO : BOOL ;	//1=APRIRE IL FRENO DI STAZIONAMENTO
END_VAR
VAR_IN_OUT
  START_ASSOLUTO : BOOL ;	//1=START POSIZIONAMENTO ASSOLUTO
  START_INCREMENTALE : BOOL ;	//1=START POSIZIONAMENTO INCREMENTALE
  START_HOME : BOOL ;	//1=START RICERCA ZERO
  START_RIPOSIZIONAMENTO : BOOL ;	//1=START POSIZIONAMENTO SU POSIZIONE INIZIALE
END_VAR
VAR
  SCELTA_BLOCCO : WORD ;
  BLOCCO_ATTUALE : WORD ;
  INVIA_JOB1 : BOOL ;	//INVIO COMANDO DI CARICA BLOCCO ASSOLUTO
  JOB1_ULTIMATO : BOOL ;	//IL NUOVO BLOCCO DI MOVIMENTO ASSOLUTO E' STATO INVIATO
  INVIA_JOB2 : BOOL ;	//INVIO COMANDO DI CARICA BLOCCO INCREMENTALE
  JOB2_ULTIMATO : BOOL ;	//IL NUOVO BLOCCO DI MOVIMENTO INCREMENTALE E' STATO INVIATO
  GIA_IN_POSIZIONE : BOOL ;	//POSIZIONAMENTO NON NECESSARIO PER ASSE GIA' IN POSIZIONE
  PACO1 : STRUCT
   PACO1_8 : BOOL ;	//1=MARCIA A IMPULSI 1
   PACO1_9 : BOOL ;	//1=MARCIA 1 IMPULSI 2
   PACO1_10 : BOOL ;	//1=ABILITA IL COMANDO (DA METTERE A 1 QUANDO PAST1.9=1)
   PACO1_11 : BOOL ;	//1=AVVIA IL RIFERIMENTO DELL'ASSE
   PACO1_12 : BOOL ;	//RISERVATO
   PACO1_13 : BOOL ;	//1=CAMBIO BLOCCO ESTERNO
   PACO1_14 : BOOL ;	//RISERVATO
   PACO1_15 : BOOL ;	//RISERVATO
   PACO1_0 : BOOL ;	//1=INSERITO 0=DISINSERITO
   PACO1_1 : BOOL ;	//1=INSERITO 0=DISINSERITO
   PACO1_2 : BOOL ;	//1=INSERITO 0=DISINSERITO
   PACO1_3 : BOOL ;	//0=BLOCCO IMPULSI (IL MOTORE SI FERMA PER INERZIA)
   PACO1_4 : BOOL ;	//1=OK 0=STOP ASSE E CANCELLAZIONE PERCORSO RESISDUO
   PACO1_5 : BOOL ;	//1=OK 0=STOP ASSE E ULTIMAZIONE MOVIMENTO CON FRONTE 0-->1
   PACO1_6 : BOOL ;	//0-->1=ATTIVARE L'ORDINE DI SPOSTAMENTO
   PACO1_7 : BOOL ;	//1=TACITAZIONE ALLARME
  END_STRUCT ;
  PAST1 : STRUCT
   PAST1_8 : BOOL ;	//1=NESSUN ERRORE D'INSEGUIMENTO
   PAST1_9 : BOOL ;	//1=SLAVE OK E PRONTO A RICEVERE COMANDI
   PAST1_10 : BOOL ;	//1=POSIZIONE RAGGIUNTA
   PAST1_11 : BOOL ;	//1=ASSE RIFERITO
   PAST1_12 : BOOL ;	//1=POSIZIONAMENTO IN CORSO
   PAST1_13 : BOOL ;	//1=MOTORE FERMO
   PAST1_14 : BOOL ;	//RISERVATO
   PAST1_15 : BOOL ;	//RISERVATO
   PAST1_0 : BOOL ;	//1=PRONTO ALL'INSERZIONE
   PAST1_1 : BOOL ;	//1=PRONTO AL FUNZIONAMENTO
   PAST1_2 : BOOL ;	//STATO ABILITAZIONE REGOLATORE
   PAST1_3 : BOOL ;	//1=PRESEZA GUASTI
   PAST1_4 : BOOL ;	//1=DISINSERIMENTO 2 ASSENTE
   PAST1_5 : BOOL ;	//1=DISINSERIMENTO 3 ASSENTE
   PAST1_6 : BOOL ;	//1=BLOCCO ALL'INSERZIONE
   PAST1_7 : BOOL ;	//1=PRESENZA AVVISI
  END_STRUCT ;
  DIGin : STRUCT
   DIGin_8 : BOOL ;
   DIGin_9 : BOOL ;
   DIGin_10 : BOOL ;
   DIGin_11 : BOOL ;
   DIGin_12 : BOOL ;
   DIGin_13 : BOOL ;
   DIGin_14 : BOOL ;
   DIGin_15 : BOOL ;
   DIGin_0 : BOOL ;	//1=ASSE SU CAMMA DI HOME
   DIGin_1 : BOOL ;	//1=ASSE SU EXTRACORSA NEGATIVO
   DIGin_2 : BOOL ;	//1=ASSE SU EXTRACORSA POSITIVO
   DIGin_3 : BOOL ;
   DIGin_4 : BOOL ;
   DIGin_5 : BOOL ;
   DIGin_6 : BOOL ;
   DIGin_7 : BOOL ;
  END_STRUCT ;
  AUX1 : BOOL ;	//APPOGGIO PER FRONTE
  AUX2 : BOOL ;	//APPOGGIO PER FRONTE
  AUX3 : BOOL ;	//APPOGGIO PER FRONTE
  AUX4 : BOOL ;	//APPOGGIO PER FRONTE
  AUX5 : BOOL ;	//APPOGGIO PER FRONTE
  AUX6 : BOOL ;	//APPOGGIO PER FRONTE
  AUX7 : BOOL ;	//APPOGGIO PER FRONTE
  VERIFICA_SPOSTAMENTO : DINT ;	//DIFFERENZA TRA TARGET E POSIZIONE ATTUALE
  PAST2 : STRUCT
   PAST2_8 : BOOL ;	//1=TACITARE IL GUASTO 608
   PAST2_9 : BOOL ;	//1=ATTUALE MOTORE 1.SEGNALE
   PAST2_10 : BOOL ;	//1=ATTUALE MOTORE 2.SEGNALE
   PAST2_11 : BOOL ;	//1=RISERVATO
   PAST2_12 : BOOL ;
   PAST2_13 : BOOL ;
   PAST2_14 : BOOL ;
   PAST2_15 : BOOL ;
   PAST2_0 : BOOL ;
   PAST2_1 : BOOL ;
   PAST2_2 : BOOL ;
   PAST2_3 : BOOL ;	//PRIMO FILTRO DEL RIFERIMENTO ATTIVO
   PAST2_4 : BOOL ;	//BLOCCO DELL'INTEGRATORE NEL REGOLATORE DI VELOCITA'
   PAST2_5 : BOOL ;	//APRIRE IL FRENO DI STAZIONAMENTO
   PAST2_6 : BOOL ;	//BLOCCO DELL'INTEGRATORE NEL REGOLATORE DI VELOCITA'
   PAST2_7 : BOOL ;	//SCELTO L'ASSE IN PARCHEGGIO
  END_STRUCT ;
  POS_PAST : STRUCT
   POS_PAST_0 : BOOL ;	//FUNZIONAMENTO A SEGUIRE
   POS_PAST_1 : BOOL ;	//LIMITAZIONE DELLA VELOCITA' LINEARE ATTIVA
   POS_PAST_2 : BOOL ;	//C'E' IL RIFERIMENTO
   POS_PAST_3 : BOOL ;	//BIT DI FUNZIONE
   POS_PAST_4 : BOOL ;	//L'ASSE SI SPOSTA IN AVANTI
   POS_PAST_5 : BOOL ;	//L'ASSE SI SPOSTA INDIETRO
   POS_PAST_6 : BOOL ;	//FINECORSA SOFTWARE MENO
   POS_PAST_7 : BOOL ;	//FINECORSA SOFTWARE PIU'
   POS_PAST_8 : BOOL ;	//SEGNALE D'INSERZIONE DELLA CAMMA 1
   POS_PAST_9 : BOOL ;	//SEGNALE D'INSERZIONE DELLA CAMMA 2
   POS_PAST_10 : BOOL ;	//USCITA DIRETTA 1 CON IL BLOCCO DI SPOSTAMENTO
   POS_PAST_11 : BOOL ;	//USCITA DIRETTA 2 CON IL BLOCCO DI SPOSTAMENTO
   POS_PAST_12 : BOOL ;	//RISERVATO
   POS_PAST_13 : BOOL ;	//RISERVATO
   POS_PAST_14 : BOOL ;	//RISERVATO
   POS_PAST_15 : BOOL ;	//RISERVATO
  END_STRUCT ;
END_VAR
BEGIN
NETWORK
TITLE = AGGIORNAMENTO IMMAGINE INGRESSI
      L     #INDIRIZZO_INIZIALE_E_A;
      L     8;
      +I;
      SLD   3;
      T     "MD100";
      L     PIW ["MD100"];	//;PAST1
      T     DIW 52;
      L     "MD100";
      SRW   3;
      L     2;
      +D;
      SLW   3;
      T     "MD100";
//;
      L     PIW ["MD100"];	//;BLOCCO ATTUALE
      T     #BLOCCO_ATTUALE;
      L     "MD100";
      SRW   3;
      L     2;
      +D;
      SLW   3;
      T     "MD100";
//;
      L     PIW ["MD100"];	//;POS PAST
      T     DIW 64;
      L     "MD100";
      SRW   3;
      L     2;
      +D;
      SLW   3;
      T     "MD100";
//;
      L     PIW ["MD100"];	//;PAST 2
      T     DIW 62;
      L     "MD100";
      SRW   3;
      L     2;
      +D;
      SLW   3;
      T     "MD100";
//;
      L     PID ["MD100"];	//; POSIZIONE ATTUALE
      T     #POSIZIONE_ATTUALE;
      L     "MD100";
      SRW   3;
      L     4;
      +D;
      SLW   3;
      T     "MD100";
//;
      L     PIW ["MD100"];	//;INGRESSI DIGITALI
      T     DIW 54;
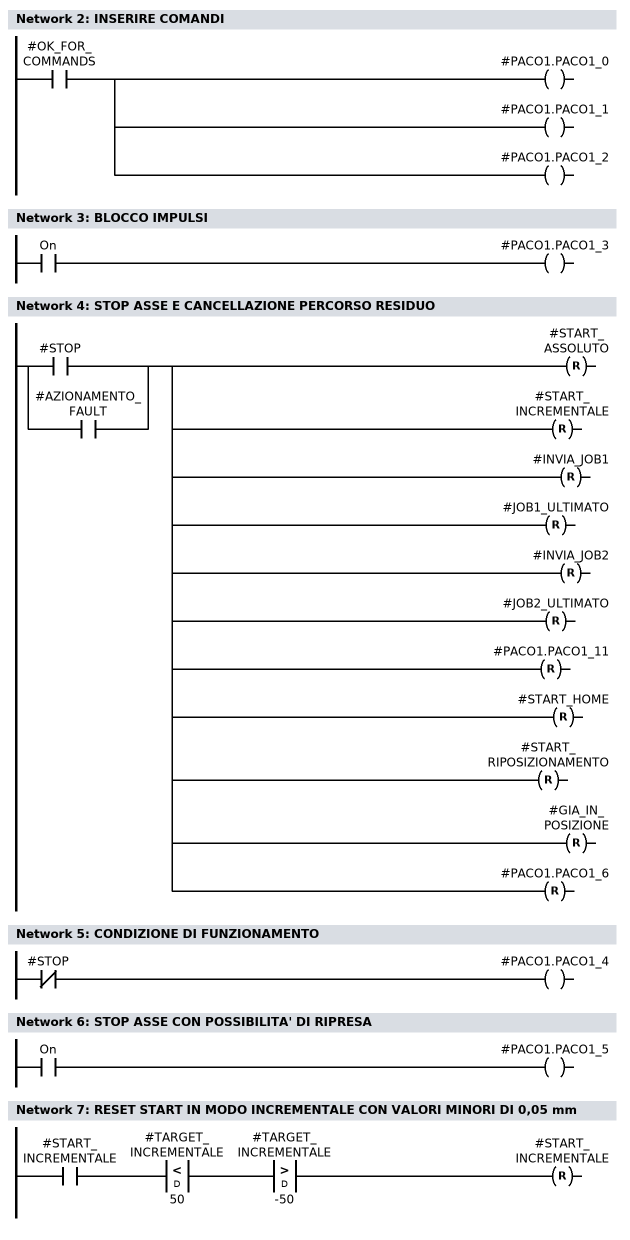
NETWORK
TITLE = INSERIRE COMANDI
      A     #OK_FOR_COMMANDS;
      =     #PACO1.PACO1_0;
      =     #PACO1.PACO1_1;
      =     #PACO1.PACO1_2;
NETWORK
TITLE = BLOCCO IMPULSI
      A     "On";
      =     #PACO1.PACO1_3;
NETWORK
TITLE = STOP ASSE E CANCELLAZIONE PERCORSO RESIDUO
      O     #STOP;
      O     #AZIONAMENTO_FAULT;
      R     #START_ASSOLUTO;
      R     #START_INCREMENTALE;
      R     #INVIA_JOB1;
      R     #JOB1_ULTIMATO;
      R     #INVIA_JOB2;
      R     #JOB2_ULTIMATO;
      R     #PACO1.PACO1_11;
      R     #START_HOME;
      R     #START_RIPOSIZIONAMENTO;
      R     #GIA_IN_POSIZIONE;
      R     #PACO1.PACO1_6;
NETWORK
TITLE = CONDIZIONE DI FUNZIONAMENTO
      AN    #STOP;
      =     #PACO1.PACO1_4;
NETWORK
TITLE = STOP ASSE CON POSSIBILITA' DI RIPRESA 
      A     "On";
      =     #PACO1.PACO1_5;
NETWORK
TITLE = RESET START IN MODO INCREMENTALE CON VALORI MINORI DI 0,05 mm
      A     #START_INCREMENTALE;
      A(;
      L     #TARGET_INCREMENTALE;
      L     50;
      <D;
      );
      A(;
      L     #TARGET_INCREMENTALE;
      L     -50;
      >D;
      );
      R     #START_INCREMENTALE;
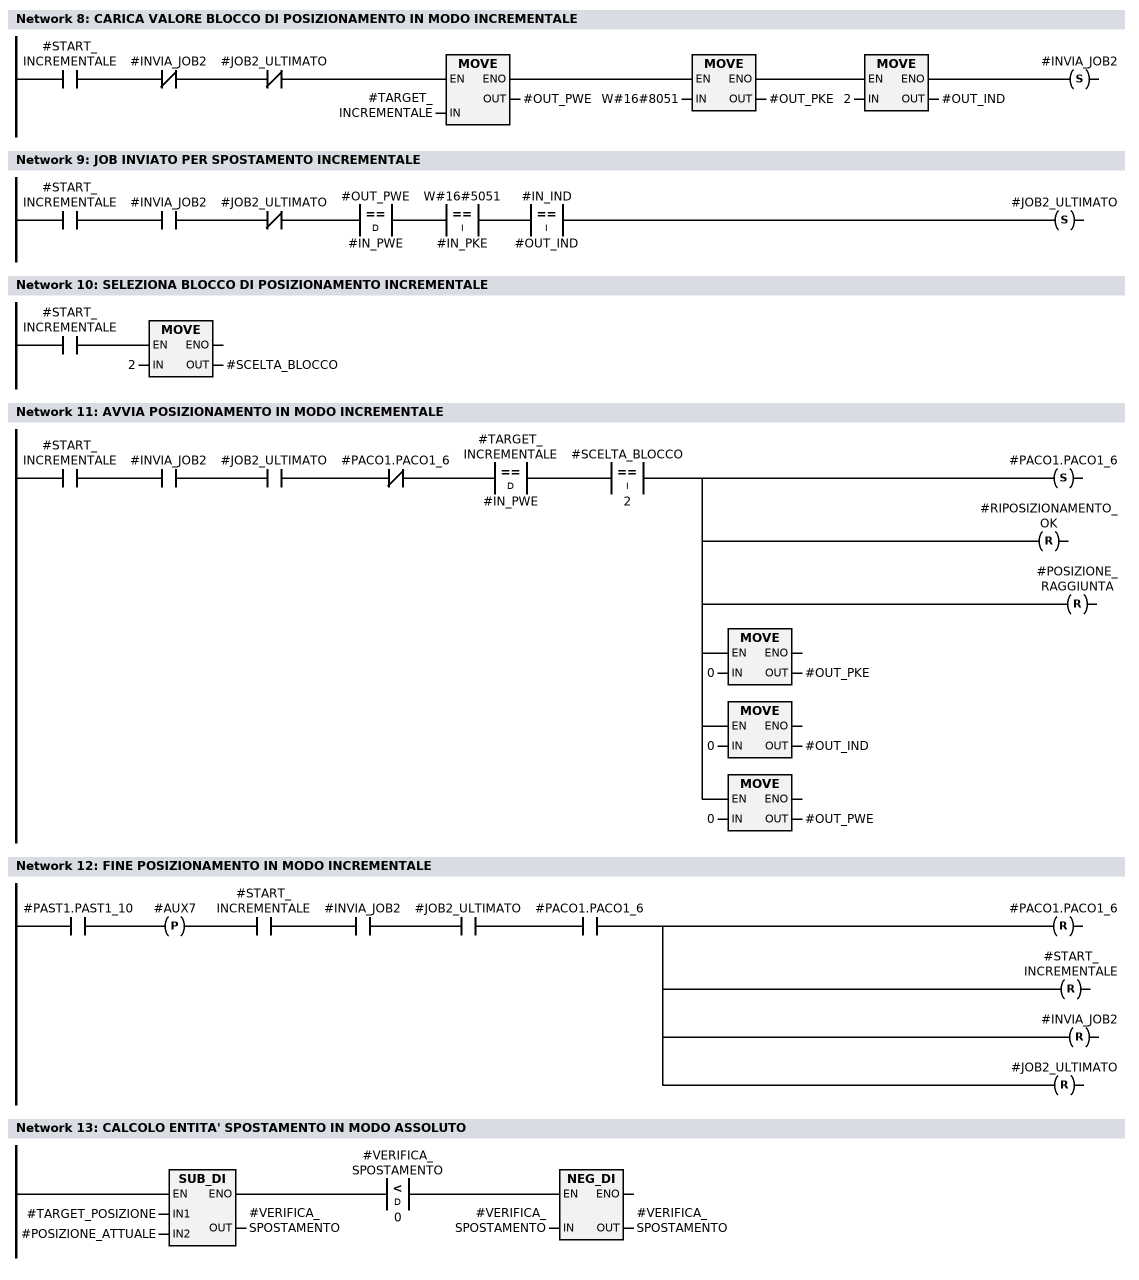
NETWORK
TITLE = CARICA VALORE BLOCCO DI POSIZIONAMENTO IN MODO INCREMENTALE
      A(;
      A(;
      A     #START_INCREMENTALE;
      AN    #INVIA_JOB2;
      AN    #JOB2_ULTIMATO;
      JNB   _001;
      L     #TARGET_INCREMENTALE;
      T     #OUT_PWE;
      SET;
      SAVE;
      CLR;
_001: A     BR;
      );
      JNB   _002;
      L     W#16#8051;
      T     #OUT_PKE;
      SET;
      SAVE;
      CLR;
_002: A     BR;
      );
      JNB   _003;
      L     2;
      T     #OUT_IND;
      SET;
      SAVE;
      CLR;
_003: A     BR;
      S     #INVIA_JOB2;
NETWORK
TITLE = JOB INVIATO PER SPOSTAMENTO INCREMENTALE
      A     #START_INCREMENTALE;
      A     #INVIA_JOB2;
      AN    #JOB2_ULTIMATO;
      A(;
      L     #OUT_PWE;
      L     #IN_PWE;
      ==D;
      );
      A(;
      L     W#16#5051;
      L     #IN_PKE;
      ==I;
      );
      A(;
      L     #IN_IND;
      L     #OUT_IND;
      ==I;
      );
      S     #JOB2_ULTIMATO;
NETWORK
TITLE = SELEZIONA BLOCCO DI POSIZIONAMENTO INCREMENTALE
      A     #START_INCREMENTALE;
      JNB   _004;
      L     2;
      T     #SCELTA_BLOCCO;
_004: NOP   0;
NETWORK
TITLE = AVVIA POSIZIONAMENTO IN MODO INCREMENTALE
      A     #START_INCREMENTALE;
      A     #INVIA_JOB2;
      A     #JOB2_ULTIMATO;
      AN    #PACO1.PACO1_6;
      A(;
      L     #TARGET_INCREMENTALE;
      L     #IN_PWE;
      ==D;
      );
      A(;
      L     #SCELTA_BLOCCO;
      L     2;
      ==I;
      );
      =     L 0.0;
      A     L 0.0;
      BLD   102;
      S     #PACO1.PACO1_6;
      A     L 0.0;
      BLD   102;
      R     #RIPOSIZIONAMENTO_OK;
      A     L 0.0;
      BLD   102;
      R     #POSIZIONE_RAGGIUNTA;
      A     L 0.0;
      JNB   _005;
      L     0;
      T     #OUT_PKE;
_005: NOP   0;
      A     L 0.0;
      JNB   _006;
      L     0;
      T     #OUT_IND;
_006: NOP   0;
      A     L 0.0;
      JNB   _007;
      L     0;
      T     #OUT_PWE;
_007: NOP   0;
NETWORK
TITLE = FINE POSIZIONAMENTO IN MODO INCREMENTALE
      A     #PAST1.PAST1_10;
      FP    #AUX7;
      A     #START_INCREMENTALE;
      A     #INVIA_JOB2;
      A     #JOB2_ULTIMATO;
      A     #PACO1.PACO1_6;
      R     #PACO1.PACO1_6;
      R     #START_INCREMENTALE;
      R     #INVIA_JOB2;
      R     #JOB2_ULTIMATO;
NETWORK
TITLE = CALCOLO ENTITA' SPOSTAMENTO IN MODO ASSOLUTO
      A(;
      L     #TARGET_POSIZIONE;
      L     #POSIZIONE_ATTUALE;
      -D;
      T     #VERIFICA_SPOSTAMENTO;
      AN    OV;
      SAVE;
      CLR;
      A     BR;
      );
      A(;
      L     #VERIFICA_SPOSTAMENTO;
      L     0;
      <D;
      );
      JNB   _008;
      L     #VERIFICA_SPOSTAMENTO;
      NEGD;
      T     #VERIFICA_SPOSTAMENTO;
_008: NOP   0;
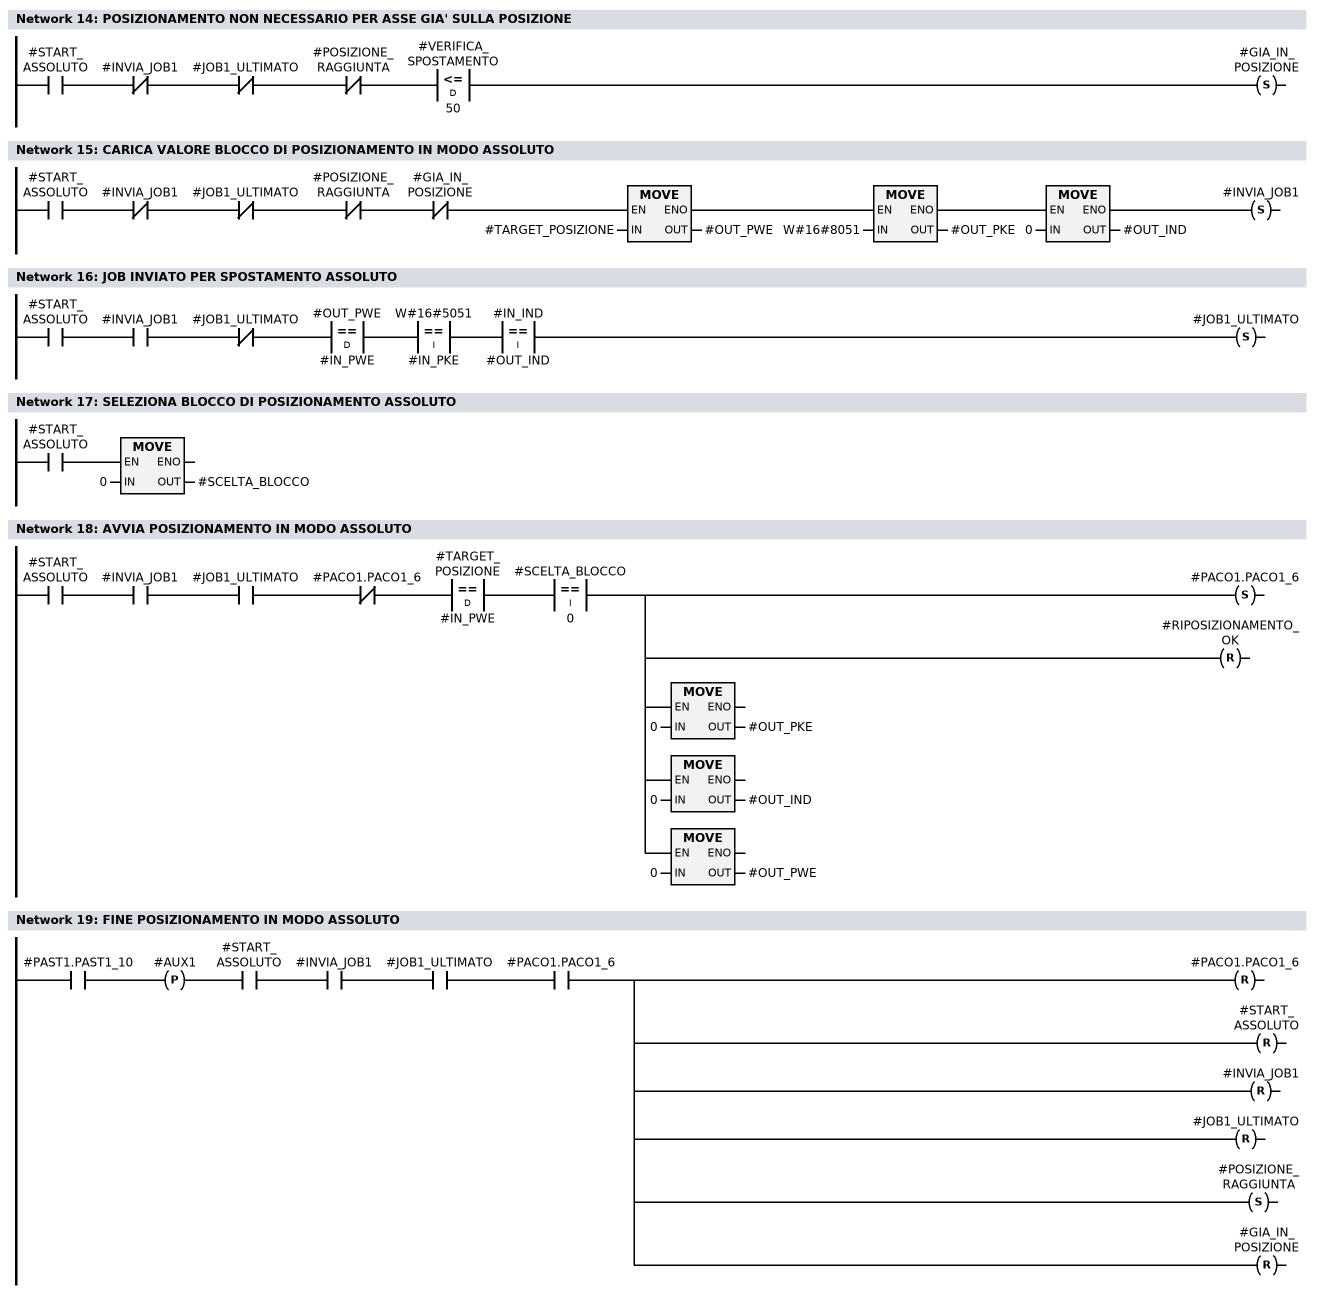
NETWORK
TITLE = POSIZIONAMENTO NON NECESSARIO PER ASSE GIA' SULLA POSIZIONE
      A     #START_ASSOLUTO;
      AN    #INVIA_JOB1;
      AN    #JOB1_ULTIMATO;
      AN    #POSIZIONE_RAGGIUNTA;
      A(;
      L     #VERIFICA_SPOSTAMENTO;
      L     50;
      <=D;
      );
      S     #GIA_IN_POSIZIONE;
NETWORK
TITLE = CARICA VALORE BLOCCO DI POSIZIONAMENTO IN MODO ASSOLUTO
      A(;
      A(;
      A     #START_ASSOLUTO;
      AN    #INVIA_JOB1;
      AN    #JOB1_ULTIMATO;
      AN    #POSIZIONE_RAGGIUNTA;
      AN    #GIA_IN_POSIZIONE;
      JNB   _009;
      L     #TARGET_POSIZIONE;
      T     #OUT_PWE;
      SET;
      SAVE;
      CLR;
_009: A     BR;
      );
      JNB   _00a;
      L     W#16#8051;
      T     #OUT_PKE;
      SET;
      SAVE;
      CLR;
_00a: A     BR;
      );
      JNB   _00b;
      L     0;
      T     #OUT_IND;
      SET;
      SAVE;
      CLR;
_00b: A     BR;
      S     #INVIA_JOB1;
NETWORK
TITLE = JOB INVIATO PER SPOSTAMENTO ASSOLUTO
      A     #START_ASSOLUTO;
      A     #INVIA_JOB1;
      AN    #JOB1_ULTIMATO;
      A(;
      L     #OUT_PWE;
      L     #IN_PWE;
      ==D;
      );
      A(;
      L     W#16#5051;
      L     #IN_PKE;
      ==I;
      );
      A(;
      L     #IN_IND;
      L     #OUT_IND;
      ==I;
      );
      S     #JOB1_ULTIMATO;
NETWORK
TITLE = SELEZIONA BLOCCO DI POSIZIONAMENTO ASSOLUTO
      A     #START_ASSOLUTO;
      JNB   _00c;
      L     0;
      T     #SCELTA_BLOCCO;
_00c: NOP   0;
NETWORK
TITLE = AVVIA POSIZIONAMENTO IN MODO ASSOLUTO
      A     #START_ASSOLUTO;
      A     #INVIA_JOB1;
      A     #JOB1_ULTIMATO;
      AN    #PACO1.PACO1_6;
      A(;
      L     #TARGET_POSIZIONE;
      L     #IN_PWE;
      ==D;
      );
      A(;
      L     #SCELTA_BLOCCO;
      L     0;
      ==I;
      );
      =     L 0.0;
      A     L 0.0;
      BLD   102;
      S     #PACO1.PACO1_6;
      A     L 0.0;
      BLD   102;
      R     #RIPOSIZIONAMENTO_OK;
      A     L 0.0;
      JNB   _00d;
      L     0;
      T     #OUT_PKE;
_00d: NOP   0;
      A     L 0.0;
      JNB   _00e;
      L     0;
      T     #OUT_IND;
_00e: NOP   0;
      A     L 0.0;
      JNB   _00f;
      L     0;
      T     #OUT_PWE;
_00f: NOP   0;
NETWORK
TITLE = FINE POSIZIONAMENTO IN MODO ASSOLUTO
      A     #PAST1.PAST1_10;
      FP    #AUX1;
      A     #START_ASSOLUTO;
      A     #INVIA_JOB1;
      A     #JOB1_ULTIMATO;
      A     #PACO1.PACO1_6;
      R     #PACO1.PACO1_6;
      R     #START_ASSOLUTO;
      R     #INVIA_JOB1;
      R     #JOB1_ULTIMATO;
      S     #POSIZIONE_RAGGIUNTA;
      R     #GIA_IN_POSIZIONE;
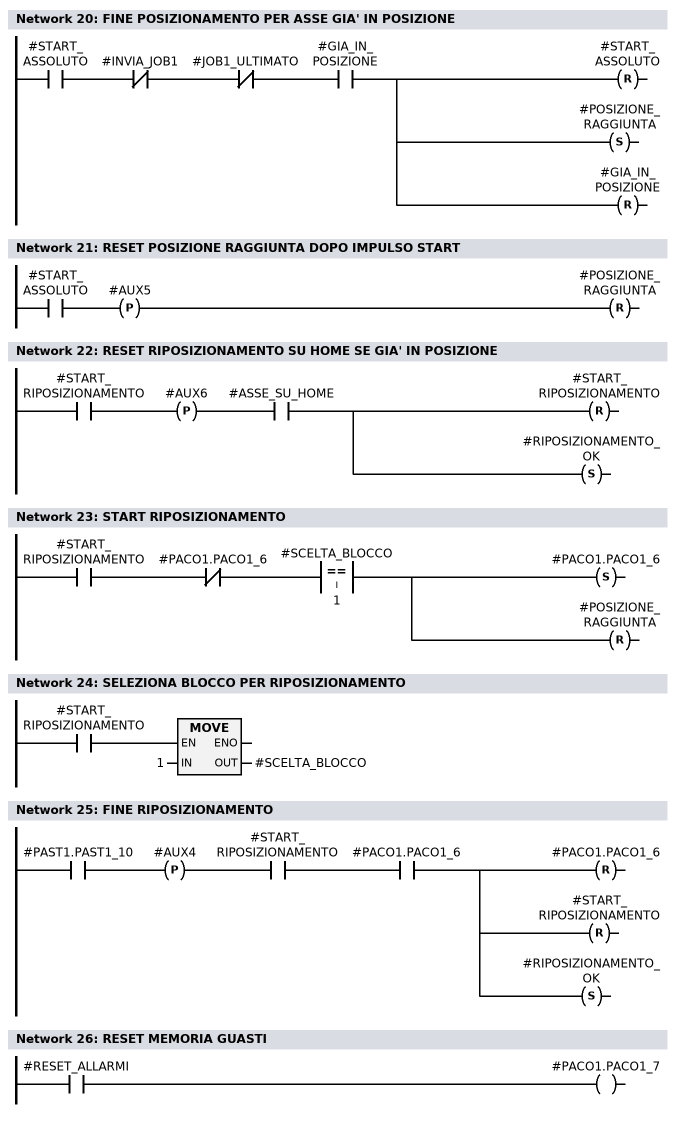
NETWORK
TITLE = FINE POSIZIONAMENTO PER ASSE GIA' IN POSIZIONE
      A     #START_ASSOLUTO;
      AN    #INVIA_JOB1;
      AN    #JOB1_ULTIMATO;
      A     #GIA_IN_POSIZIONE;
      R     #START_ASSOLUTO;
      S     #POSIZIONE_RAGGIUNTA;
      R     #GIA_IN_POSIZIONE;
NETWORK
TITLE = RESET POSIZIONE RAGGIUNTA DOPO IMPULSO START
      A     #START_ASSOLUTO;
      FP    #AUX5;
      R     #POSIZIONE_RAGGIUNTA;
NETWORK
TITLE = RESET RIPOSIZIONAMENTO SU HOME SE GIA' IN POSIZIONE
      A     #START_RIPOSIZIONAMENTO;
      FP    #AUX6;
      A     #ASSE_SU_HOME;
      R     #START_RIPOSIZIONAMENTO;
      S     #RIPOSIZIONAMENTO_OK;
NETWORK
TITLE = START RIPOSIZIONAMENTO
      A     #START_RIPOSIZIONAMENTO;
      AN    #PACO1.PACO1_6;
      A(;
      L     #SCELTA_BLOCCO;
      L     1;
      ==I;
      );
      S     #PACO1.PACO1_6;
      R     #POSIZIONE_RAGGIUNTA;
NETWORK
TITLE = SELEZIONA BLOCCO PER RIPOSIZIONAMENTO
      A     #START_RIPOSIZIONAMENTO;
      JNB   _010;
      L     1;
      T     #SCELTA_BLOCCO;
_010: NOP   0;
NETWORK
TITLE = FINE RIPOSIZIONAMENTO
      A     #PAST1.PAST1_10;
      FP    #AUX4;
      A     #START_RIPOSIZIONAMENTO;
      A     #PACO1.PACO1_6;
      R     #PACO1.PACO1_6;
      R     #START_RIPOSIZIONAMENTO;
      S     #RIPOSIZIONAMENTO_OK;
NETWORK
TITLE = RESET MEMORIA GUASTI
      A     #RESET_ALLARMI;
      =     #PACO1.PACO1_7;
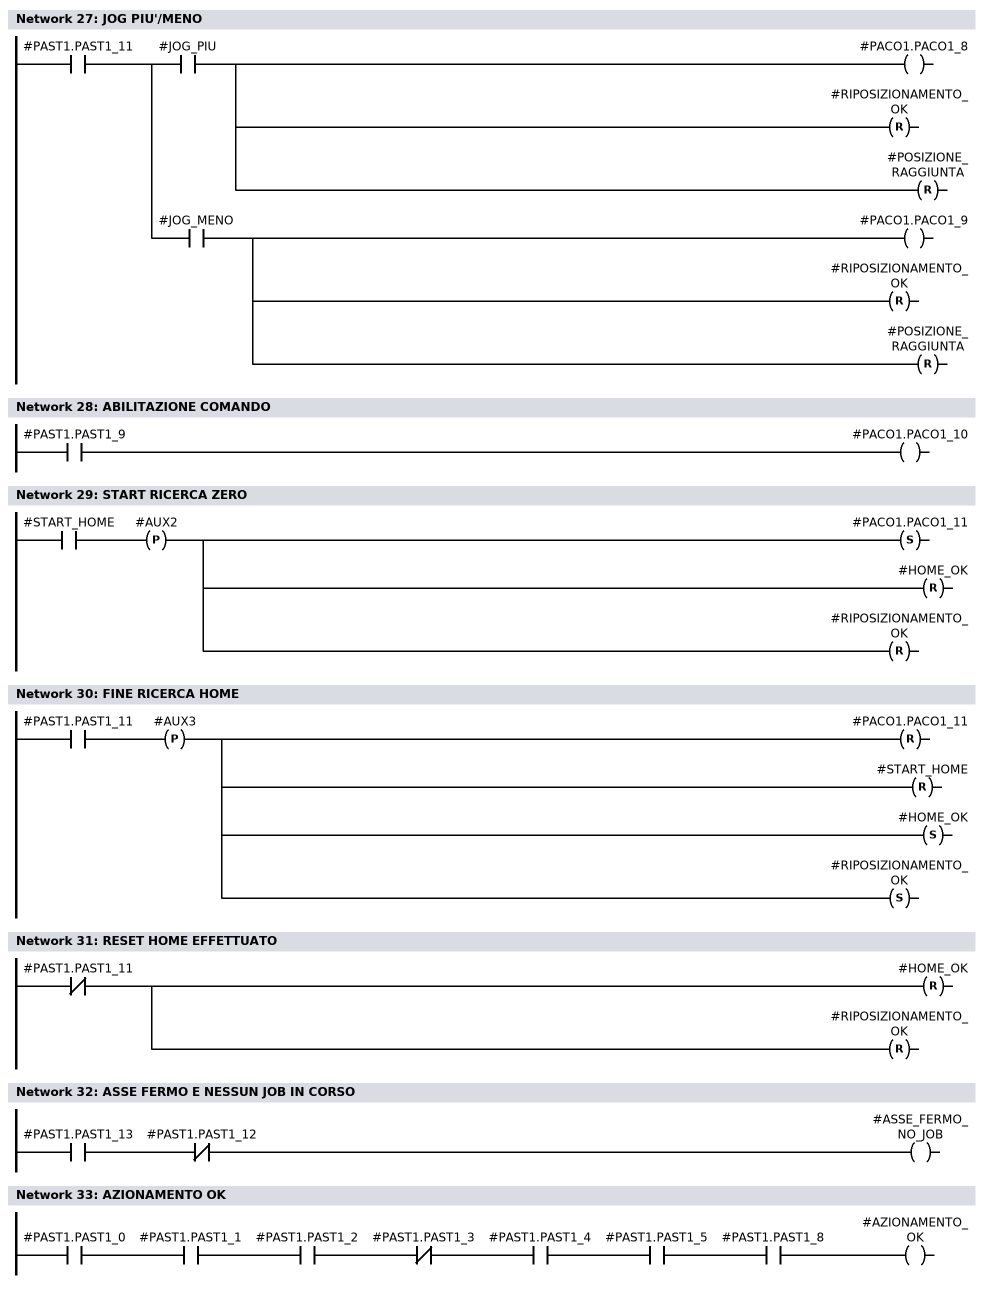
NETWORK
TITLE = JOG PIU'/MENO
      A     #PAST1.PAST1_11;
      =     L 0.0;
      A     L 0.0;
      A     #JOG_PIU;
      =     #PACO1.PACO1_8;
      R     #RIPOSIZIONAMENTO_OK;
      R     #POSIZIONE_RAGGIUNTA;
      A     L 0.0;
      A     #JOG_MENO;
      =     #PACO1.PACO1_9;
      R     #RIPOSIZIONAMENTO_OK;
      R     #POSIZIONE_RAGGIUNTA;
NETWORK
TITLE = ABILITAZIONE COMANDO
      A     #PAST1.PAST1_9;
      =     #PACO1.PACO1_10;
NETWORK
TITLE = START RICERCA ZERO
      A     #START_HOME;
      FP    #AUX2;
      S     #PACO1.PACO1_11;
      R     #HOME_OK;
      R     #RIPOSIZIONAMENTO_OK;
NETWORK
TITLE = FINE RICERCA HOME
      A     #PAST1.PAST1_11;
      FP    #AUX3;
      R     #PACO1.PACO1_11;
      R     #START_HOME;
      S     #HOME_OK;
      S     #RIPOSIZIONAMENTO_OK;
NETWORK
TITLE = RESET HOME EFFETTUATO
      AN    #PAST1.PAST1_11;
      R     #HOME_OK;
      R     #RIPOSIZIONAMENTO_OK;
NETWORK
TITLE = ASSE FERMO E NESSUN JOB IN CORSO
      A     #PAST1.PAST1_13;
      AN    #PAST1.PAST1_12;
      =     #ASSE_FERMO_NO_JOB;
NETWORK
TITLE = AZIONAMENTO OK
      A     #PAST1.PAST1_0;
      A     #PAST1.PAST1_1;
      A     #PAST1.PAST1_2;
      AN    #PAST1.PAST1_3;
      A     #PAST1.PAST1_4;
      A     #PAST1.PAST1_5;
      A     #PAST1.PAST1_8;
      =     #AZIONAMENTO_OK;
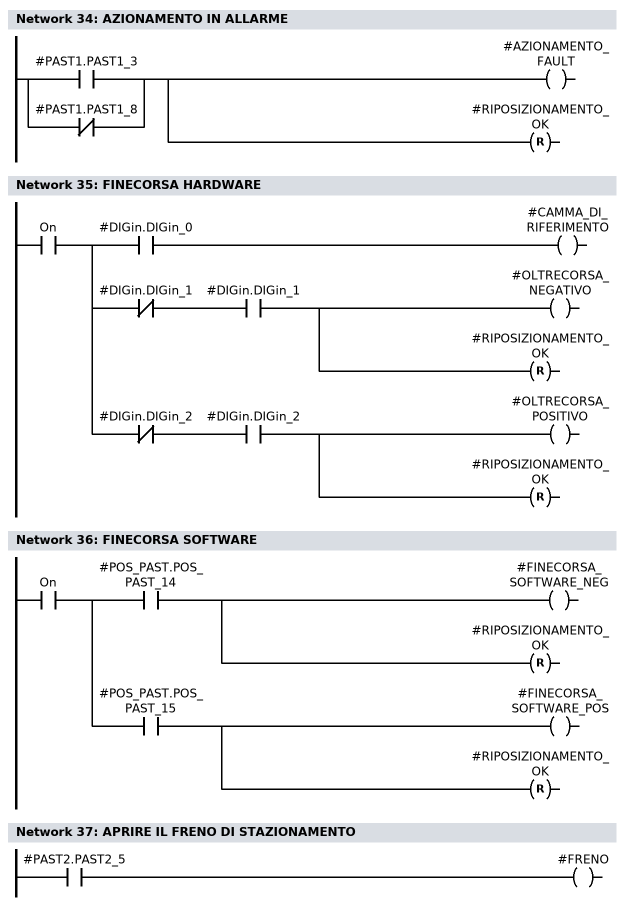
NETWORK
TITLE = AZIONAMENTO IN ALLARME
      O     #PAST1.PAST1_3;
      ON    #PAST1.PAST1_8;
      =     #AZIONAMENTO_FAULT;
      R     #RIPOSIZIONAMENTO_OK;
NETWORK
TITLE = FINECORSA HARDWARE
      A     "On";
      =     L 0.0;
      A     L 0.0;
      A     #DIGin.DIGin_0;
      =     #CAMMA_DI_RIFERIMENTO;
      A     L 0.0;
      AN    #DIGin.DIGin_1;
      A     #DIGin.DIGin_1;
      =     #OLTRECORSA_NEGATIVO;
      R     #RIPOSIZIONAMENTO_OK;
      A     L 0.0;
      AN    #DIGin.DIGin_2;
      A     #DIGin.DIGin_2;
      =     #OLTRECORSA_POSITIVO;
      R     #RIPOSIZIONAMENTO_OK;
NETWORK
TITLE = FINECORSA SOFTWARE
      A     "On";
      =     L 0.0;
      A     L 0.0;
      A     #POS_PAST.POS_PAST_14;
      =     #FINECORSA_SOFTWARE_NEG;
      R     #RIPOSIZIONAMENTO_OK;
      A     L 0.0;
      A     #POS_PAST.POS_PAST_15;
      =     #FINECORSA_SOFTWARE_POS;
      R     #RIPOSIZIONAMENTO_OK;
NETWORK
TITLE = APRIRE IL FRENO DI STAZIONAMENTO
      A     #PAST2.PAST2_5;
      =     #FRENO;
NETWORK
TITLE = AGGIORNAMENTO IMMAGINE USCITE
      L     #INDIRIZZO_INIZIALE_E_A;
      L     8;
      +I;
      SLD   3;
      T     "MD100";
      L     DIW 50;
      T     PQW ["MD100"];	//;PACO 1
      L     "MD100";
      SRW   3;
      L     2;
      +D;
      SLW   3;
      T     "MD100";
//;
      L     #SCELTA_BLOCCO;
      T     PQW ["MD100"];	//;SCELTA BLOCCO
      L     "MD100";
      SRW   3;
      L     6;
      +D;
      SLW   3;
      T     "MD100";
//;
      L     #OVERRIDE;
      T     PQW ["MD100"];	//;OVERRIDE
END_FUNCTION_BLOCK

// FC 7: know-how protected block, not included

FUNCTION "FC11 - STATUS" : VOID	// FC 11
TITLE = Sensors and proximity state
VERSION : 0.1
VAR_TEMP
  temp_INT : INT ;
END_VAR
BEGIN
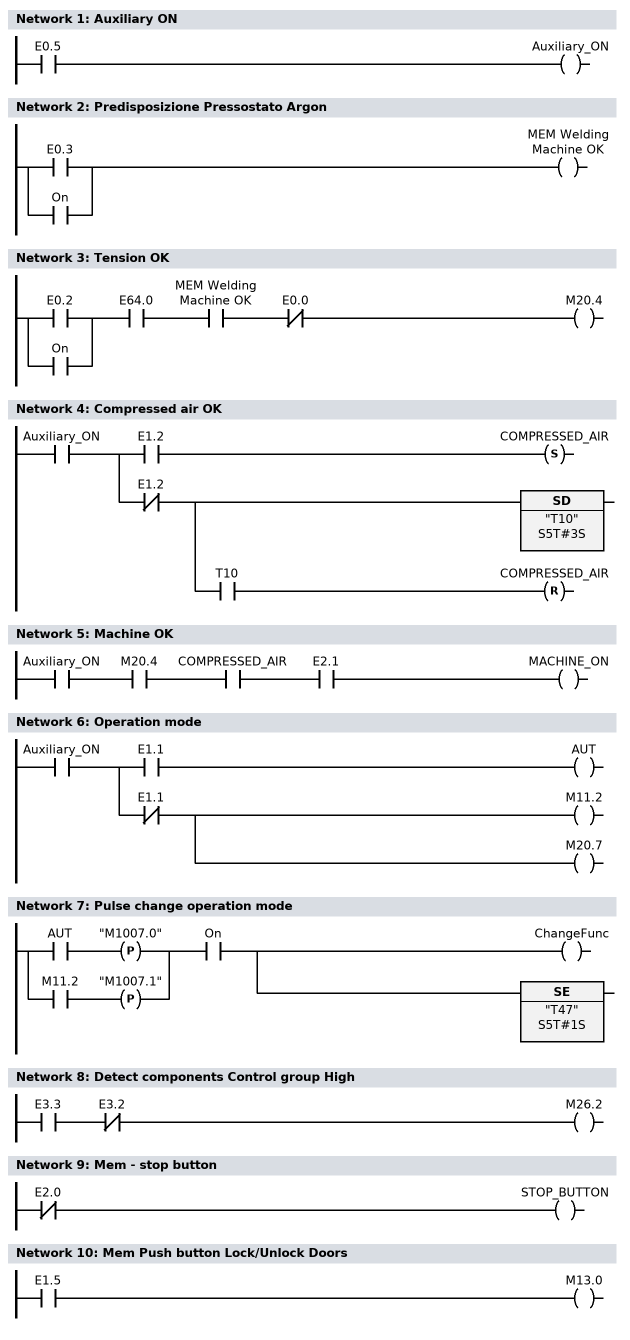
NETWORK
TITLE = Auxiliary ON
      A     "E0.5";
      =     "Auxiliary_ON";
NETWORK
TITLE = Predisposizione Pressostato Argon
      O     "E0.3";
      O     "On";
      =     "MEM Welding Machine OK";
NETWORK
TITLE = Tension OK
      A(;
      O     "E0.2";
      O     "On";
      );
      A     "E64.0";
      A     "MEM Welding Machine OK";
      AN    "E0.0";
      =     "M20.4";
NETWORK
TITLE = Compressed air OK
      A     "Auxiliary_ON";
      =     L 2.0;
      A     L 2.0;
      A     "E1.2";
      S     "COMPRESSED_AIR";
      A     L 2.0;
      AN    "E1.2";
      =     L 2.1;
      A     L 2.1;
      BLD   102;
      L     S5T#3S;
      SD    "T10";
      A     L 2.1;
      A     "T10";
      R     "COMPRESSED_AIR";
NETWORK
TITLE = Machine OK
      A     "Auxiliary_ON";
      A     "M20.4";
      A     "COMPRESSED_AIR";
      A     "E2.1";
      =     "MACHINE_ON";
NETWORK
TITLE = Operation mode
      A     "Auxiliary_ON";
      =     L 2.0;
      A     L 2.0;
      A     "E1.1";
      =     "AUT";
      A     L 2.0;
      AN    "E1.1";
      =     "M11.2";
      =     "M20.7";
NETWORK
TITLE = Pulse change operation mode
      A(;
      A     "AUT";
      FP    "M1007.0";
      O(;
      A     "M11.2";
      FP    "M1007.1";
      );
      );
      A     "On";
      =     "ChangeFunc";
      L     S5T#1S;
      SE    "T47";
NETWORK
TITLE = Detect components Control group High
      A     "E3.3";
      AN    "E3.2";
      =     "M26.2";
NETWORK
TITLE = Mem - stop button
      AN    "E2.0";
      =     "STOP_BUTTON";
NETWORK
TITLE = Mem Push button Lock/Unlock Doors
      A     "E1.5";
      =     "M13.0";
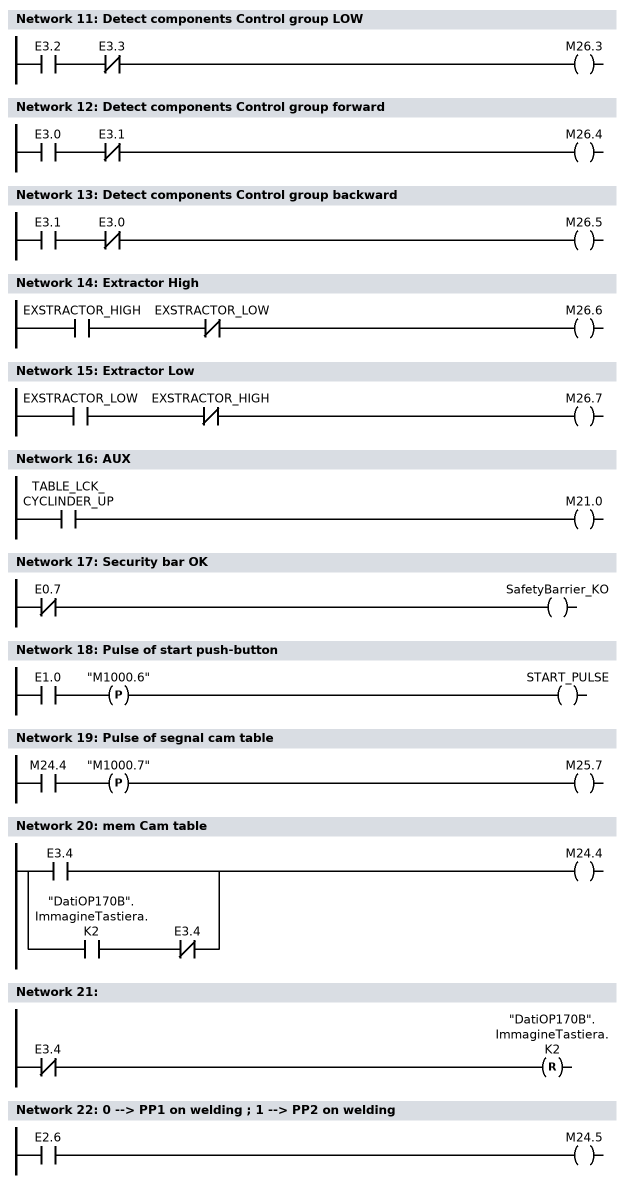
NETWORK
TITLE = Detect components Control group LOW
      A     "E3.2";
      AN    "E3.3";
      =     "M26.3";
NETWORK
TITLE = Detect components Control group forward
      A     "E3.0";
      AN    "E3.1";
      =     "M26.4";
NETWORK
TITLE = Detect components Control group backward
      A     "E3.1";
      AN    "E3.0";
      =     "M26.5";
NETWORK
TITLE = Extractor High
      A     "EXSTRACTOR_HIGH";
      AN    "EXSTRACTOR_LOW";
      =     "M26.6";
NETWORK
TITLE = Extractor Low
      A     "EXSTRACTOR_LOW";
      AN    "EXSTRACTOR_HIGH";
      =     "M26.7";
NETWORK
TITLE = AUX
      A     "TABLE_LCK_CYCLINDER_UP";
      =     "M21.0";
NETWORK
TITLE = Security bar OK
      AN    "E0.7";
      =     "SafetyBarrier_KO";
NETWORK
TITLE = Pulse of start push-button
      A     "E1.0";
      FP    "M1000.6";
      =     "START_PULSE";
NETWORK
TITLE = Pulse of segnal cam table
      A     "M24.4";
      FP    "M1000.7";
      =     "M25.7";
NETWORK
TITLE = mem Cam table
      O     "E3.4";
      O;
      A     "DatiOP170B".ImmagineTastiera.K2;
      AN    "E3.4";
      =     "M24.4";
NETWORK
TITLE =
      AN    "E3.4";
      R     "DatiOP170B".ImmagineTastiera.K2;
NETWORK
TITLE = 0 --> PP1 on welding ; 1 --> PP2 on welding
      A     "E2.6";
      =     "M24.5";
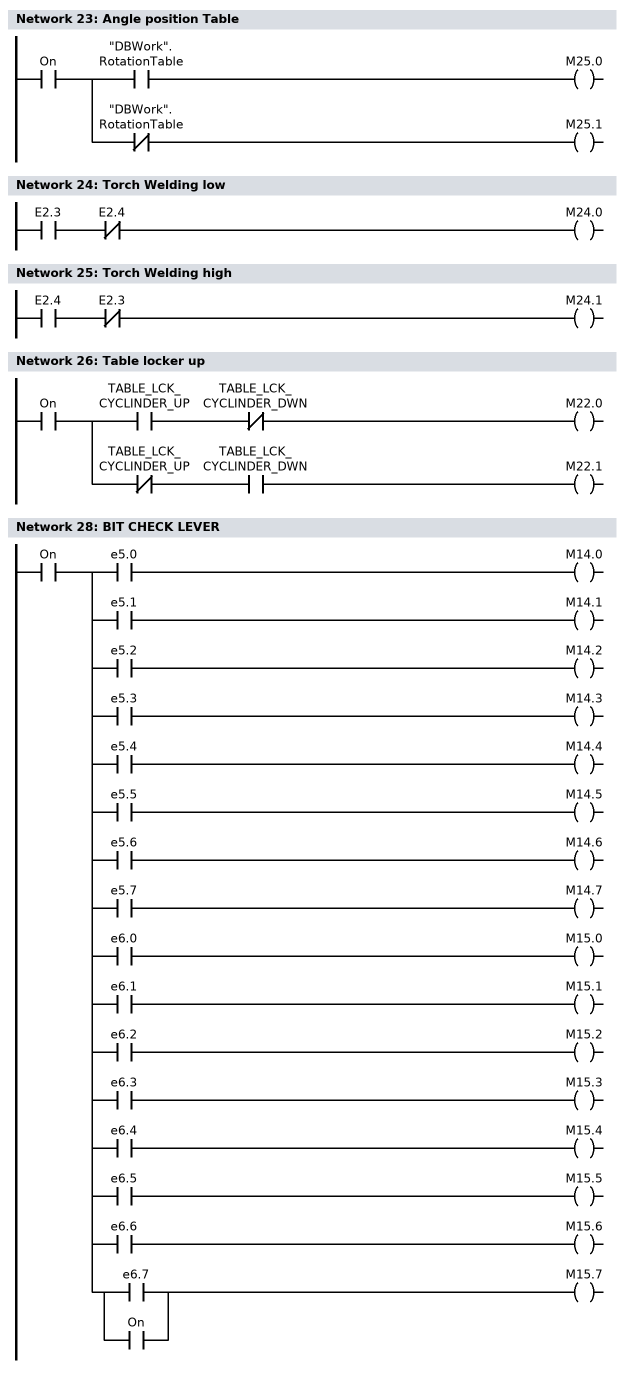
NETWORK
TITLE = Angle position Table
      A     "On";
      =     L 2.0;
      A     L 2.0;
      A     "DBWork".RotationTable;
      =     "M25.0";
      A     L 2.0;
      AN    "DBWork".RotationTable;
      =     "M25.1";
NETWORK
TITLE = Torch Welding low
      A     "E2.3";
      AN    "E2.4";
      =     "M24.0";
NETWORK
TITLE = Torch Welding high
      A     "E2.4";
      AN    "E2.3";
      =     "M24.1";
NETWORK
TITLE = Table locker up
      A     "On";
      =     L 2.0;
      A     L 2.0;
      A     "TABLE_LCK_CYCLINDER_UP";
      AN    "TABLE_LCK_CYCLINDER_DWN";
      =     "M22.0";
      A     L 2.0;
      AN    "TABLE_LCK_CYCLINDER_UP";
      A     "TABLE_LCK_CYCLINDER_DWN";
      =     "M22.1";
NETWORK
TITLE =
NETWORK
TITLE = BIT CHECK LEVER
      A     "On";
      =     L 2.0;
      A     L 2.0;
      A     "e5.0";
      =     "M14.0";
      A     L 2.0;
      A     "e5.1";
      =     "M14.1";
      A     L 2.0;
      A     "e5.2";
      =     "M14.2";
      A     L 2.0;
      A     "e5.3";
      =     "M14.3";
      A     L 2.0;
      A     "e5.4";
      =     "M14.4";
      A     L 2.0;
      A     "e5.5";
      =     "M14.5";
      A     L 2.0;
      A     "e5.6";
      =     "M14.6";
      A     L 2.0;
      A     "e5.7";
      =     "M14.7";
      A     L 2.0;
      A     "e6.0";
      =     "M15.0";
      A     L 2.0;
      A     "e6.1";
      =     "M15.1";
      A     L 2.0;
      A     "e6.2";
      =     "M15.2";
      A     L 2.0;
      A     "e6.3";
      =     "M15.3";
      A     L 2.0;
      A     "e6.4";
      =     "M15.4";
      A     L 2.0;
      A     "e6.5";
      =     "M15.5";
      A     L 2.0;
      A     "e6.6";
      =     "M15.6";
      A     L 2.0;
      A(;
      O     "e6.7";
      O     "On";
      );
      =     "M15.7";
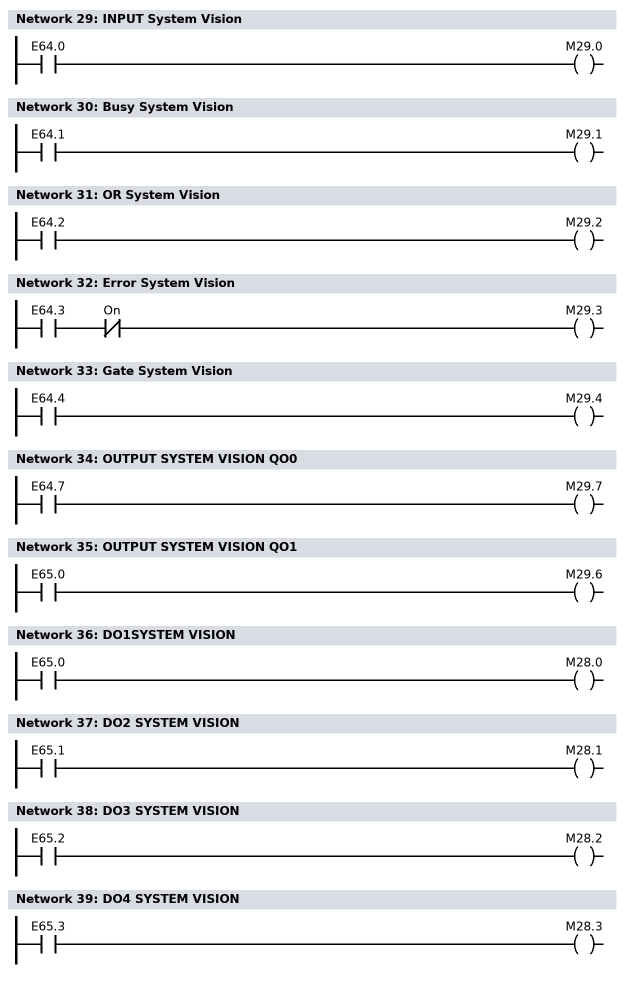
NETWORK
TITLE = INPUT System Vision 
      A     "E64.0";
      =     "M29.0";
NETWORK
TITLE = Busy System Vision
      A     "E64.1";
      =     "M29.1";
NETWORK
TITLE = OR System Vision
      A     "E64.2";
      =     "M29.2";
NETWORK
TITLE = Error System Vision
      A     "E64.3";
      AN    "On";
      =     "M29.3";
NETWORK
TITLE = Gate System Vision
      A     "E64.4";
      =     "M29.4";
NETWORK
TITLE = OUTPUT SYSTEM VISION QO0
      A     "E64.7";
      =     "M29.7";
NETWORK
TITLE = OUTPUT SYSTEM VISION QO1
      A     "E65.0";
      =     "M29.6";
NETWORK
TITLE = DO1SYSTEM VISION
      A     "E65.0";
      =     "M28.0";
NETWORK
TITLE = DO2 SYSTEM VISION
      A     "E65.1";
      =     "M28.1";
NETWORK
TITLE = DO3 SYSTEM VISION
      A     "E65.2";
      =     "M28.2";
NETWORK
TITLE = DO4 SYSTEM VISION
      A     "E65.3";
      =     "M28.3";
END_FUNCTION

FUNCTION "FC12 - GENERAL" : VOID	// FC 12
TITLE = General management
VERSION : 0.1
BEGIN
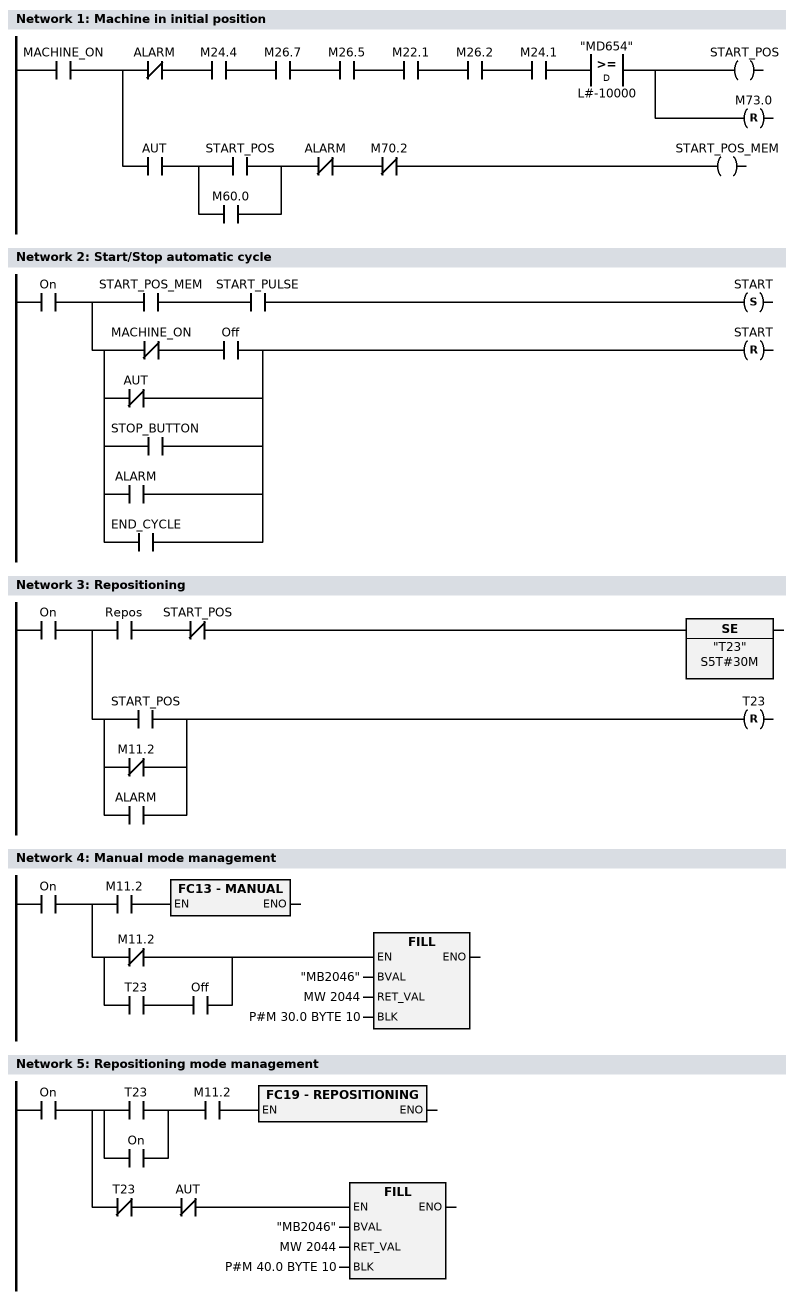
NETWORK
TITLE = Machine in initial position
      A     "MACHINE_ON";
      =     L 0.0;
      A     L 0.0;
      AN    "ALARM";
      A     "M24.4";
      A     "M26.7";
      A     "M26.5";
      A     "M22.1";
      A     "M26.2";
      A     "M24.1";
      A(;
      L     "MD654";
      L     L#-10000;
      >=D;
      );
      =     "START_POS";
      R     "M73.0";
      A     L 0.0;
      A     "AUT";
      A(;
      O     "START_POS";
      O     "M60.0";
      );
      AN    "ALARM";
      AN    "M70.2";
      =     "START_POS_MEM";
NETWORK
TITLE = Start/Stop automatic cycle
      A     "On";
      =     L 0.0;
      A     L 0.0;
      A     "START_POS_MEM";
      A     "START_PULSE";
      S     "START";
      A     L 0.0;
      A(;
      AN    "MACHINE_ON";
      A     "Off";
      ON    "AUT";
      O     "STOP_BUTTON";
      O     "ALARM";
      O     "END_CYCLE";
      );
      R     "START";
NETWORK
TITLE = Repositioning
      A     "On";
      =     L 0.0;
      A     L 0.0;
      A     "Repos";
      AN    "START_POS";
      L     S5T#30M;
      SE    "T23";
      A     L 0.0;
      A(;
      O     "START_POS";
      ON    "M11.2";
      O     "ALARM";
      );
      R     "T23";
NETWORK
TITLE = Manual mode management
      A     "On";
      =     L 0.0;
      A     L 0.0;
      A     "M11.2";
      JNB   _001;
      CALL  "FC13 - MANUAL";
_001: NOP   0;
      A     L 0.0;
      A(;
      ON    "M11.2";
      O;
      A     "T23";
      A     "Off";
      );
      JNB   _002;
      CALL  "FILL" (
           BVAL                     := "MB2046",
           RET_VAL                  := MW 2044,
           BLK                      := P#M 30.0 BYTE 10);
_002: NOP   0;
NETWORK
TITLE = Repositioning mode management
      A     "On";
      =     L 0.0;
      A     L 0.0;
      A(;
      O     "T23";
      O     "On";
      );
      A     "M11.2";
      JNB   _003;
      CALL  "FC19 - REPOSITIONING";
_003: NOP   0;
      A     L 0.0;
      AN    "T23";
      AN    "AUT";
      JNB   _004;
      CALL  "FILL" (
           BVAL                     := "MB2046",
           RET_VAL                  := MW 2044,
           BLK                      := P#M 40.0 BYTE 10);
_004: NOP   0;
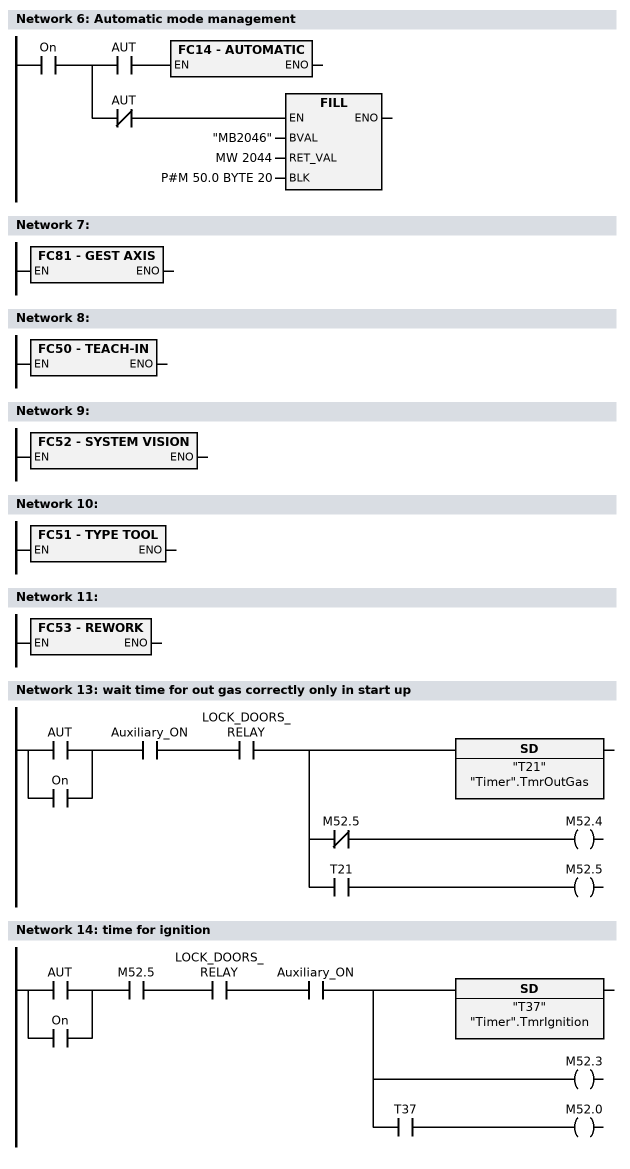
NETWORK
TITLE = Automatic mode management
//reset axis mouvement
      A     "On";
      =     L 0.0;
      A     L 0.0;
      A     "AUT";
      JNB   _005;
      CALL  "FC14 - AUTOMATIC";
_005: NOP   0;
      A     L 0.0;
      AN    "AUT";
      JNB   _006;
      CALL  "FILL" (
           BVAL                     := "MB2046",
           RET_VAL                  := MW 2044,
           BLK                      := P#M 50.0 BYTE 20);
_006: NOP   0;
NETWORK
TITLE =
      CALL  "FC81 - GEST AXIS";
      NOP   0;
NETWORK
TITLE =
      CALL  "FC50 - TEACH-IN";
      NOP   0;
NETWORK
TITLE =
      CALL  "FC52 - SYSTEM VISION";
      NOP   0;
NETWORK
TITLE =
//Controllo il tipo di portapezzo e carico i relativi dati
      CALL  "FC51 - TYPE TOOL";
      NOP   0;
NETWORK
TITLE =
      CALL  "FC53 - REWORK";
      NOP   0;
NETWORK
TITLE =
NETWORK
TITLE = wait time for out gas correctly only in start up 
//AUT - Tempo di attesa per avere gas in circolo e la torcia in temp
      A(;
      O     "AUT";
      O     "On";
      );
      A     "Auxiliary_ON";
      A     "LOCK_DOORS_RELAY";
      =     L 0.0;
      A     L 0.0;
      BLD   102;
      L     "Timer".TmrOutGas;
      SD    "T21";
      A     L 0.0;
      AN    "M52.5";
      =     "M52.4";
      A     L 0.0;
      A     "T21";
      =     "M52.5";
NETWORK
TITLE = time for ignition
      A(;
      O     "AUT";
      O     "On";
      );
      A     "M52.5";
      A     "LOCK_DOORS_RELAY";
      A     "Auxiliary_ON";
      =     L 0.0;
      A     L 0.0;
      BLD   102;
      L     "Timer".TmrIgnition;
      SD    "T37";
      A     L 0.0;
      BLD   102;
      =     "M52.3";
      A     L 0.0;
      A     "T37";
      =     "M52.0";
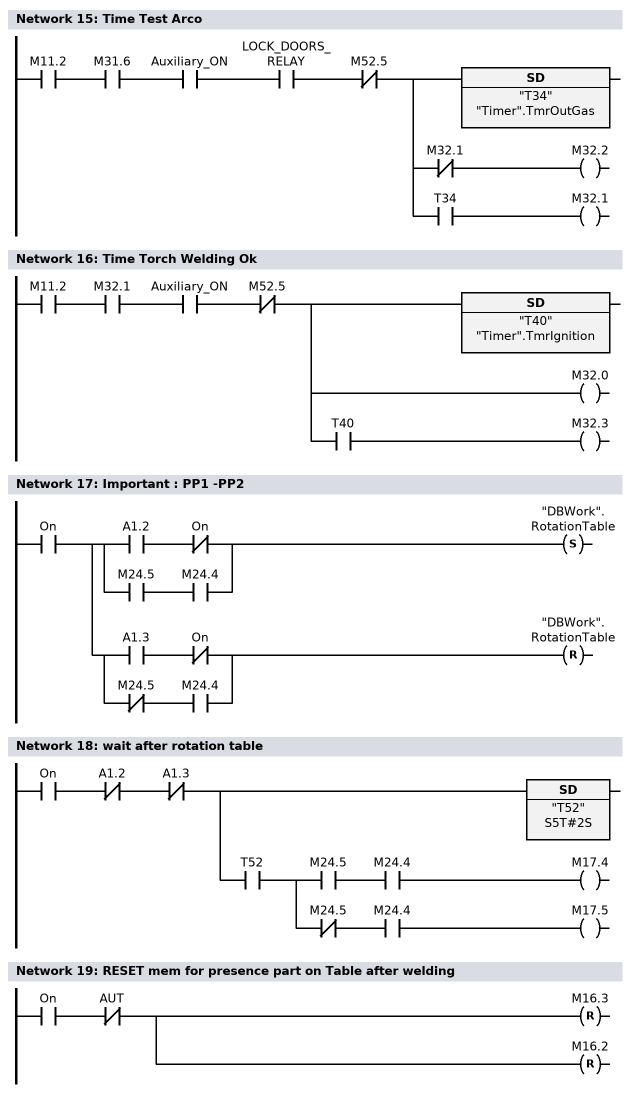
NETWORK
TITLE = Time Test Arco
//Test Arco Gas in Manuale
      A     "M11.2";
      A     "M31.6";
      A     "Auxiliary_ON";
      A     "LOCK_DOORS_RELAY";
      AN    "M52.5";
      =     L 0.0;
      A     L 0.0;
      BLD   102;
      L     "Timer".TmrOutGas;
      SD    "T34";
      A     L 0.0;
      AN    "M32.1";
      =     "M32.2";
      A     L 0.0;
      A     "T34";
      =     "M32.1";
NETWORK
TITLE = Time Torch Welding Ok
//Accensione Torcia in Manuale: per arrivare in Temp
      A     "M11.2";
      A     "M32.1";
      A     "Auxiliary_ON";
      AN    "M52.5";
      =     L 0.0;
      A     L 0.0;
      BLD   102;
      L     "Timer".TmrIgnition;
      SD    "T40";
      A     L 0.0;
      BLD   102;
      =     "M32.0";
      A     L 0.0;
      A     "T40";
      =     "M32.3";
NETWORK
TITLE = Important : PP1 -PP2 
      A     "On";
      =     L 0.0;
      A     L 0.0;
      A(;
      A     "A1.2";
      AN    "On";
      O;
      A     "M24.5";
      A     "M24.4";
      );
      S     "DBWork".RotationTable;
      A     L 0.0;
      A(;
      A     "A1.3";
      AN    "On";
      O;
      AN    "M24.5";
      A     "M24.4";
      );
      R     "DBWork".RotationTable;
NETWORK
TITLE = wait after rotation table
      A     "On";
      AN    "A1.2";
      AN    "A1.3";
      =     L 0.0;
      A     L 0.0;
      BLD   102;
      L     S5T#2S;
      SD    "T52";
      A     L 0.0;
      A     "T52";
      =     L 0.1;
      A     L 0.1;
      A     "M24.5";
      A     "M24.4";
      =     "M17.4";
      A     L 0.1;
      AN    "M24.5";
      A     "M24.4";
      =     "M17.5";
NETWORK
TITLE = RESET mem for presence part on Table after welding
      A     "On";
      AN    "AUT";
      R     "M16.3";
      R     "M16.2";
END_FUNCTION

FUNCTION "FC13 - MANUAL" : VOID	// FC 13
TITLE = Manual commands
VERSION : 0.1
BEGIN
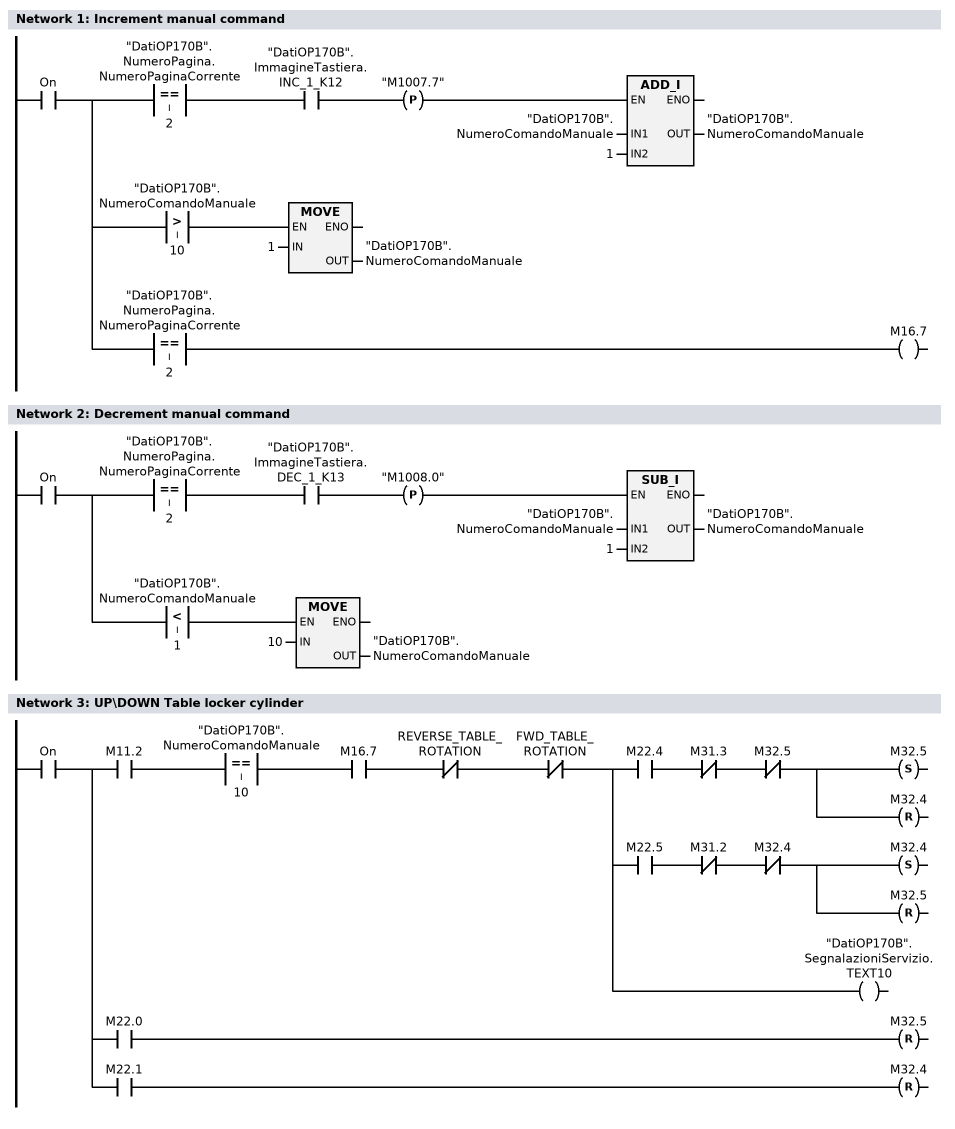
NETWORK
TITLE = Increment manual command
      A     "On";
      =     L 1.0;
      A     L 1.0;
      A(;
      L     "DatiOP170B".NumeroPagina.NumeroPaginaCorrente;
      L     2;
      ==I;
      );
      A     "DatiOP170B".ImmagineTastiera.INC_1_K12;
      FP    "M1007.7";
      JNB   _001;
      L     "DatiOP170B".NumeroComandoManuale;
      L     1;
      +I;
      T     "DatiOP170B".NumeroComandoManuale;
_001: NOP   0;
      A     L 1.0;
      A(;
      L     "DatiOP170B".NumeroComandoManuale;
      L     10;
      >I;
      );
      JNB   _002;
      L     1;
      T     "DatiOP170B".NumeroComandoManuale;
_002: NOP   0;
      A     L 1.0;
      A(;
      L     "DatiOP170B".NumeroPagina.NumeroPaginaCorrente;
      L     2;
      ==I;
      );
      =     "M16.7";
NETWORK
TITLE = Decrement manual command
      A     "On";
      =     L 1.0;
      A     L 1.0;
      A(;
      L     "DatiOP170B".NumeroPagina.NumeroPaginaCorrente;
      L     2;
      ==I;
      );
      A     "DatiOP170B".ImmagineTastiera.DEC_1_K13;
      FP    "M1008.0";
      JNB   _003;
      L     "DatiOP170B".NumeroComandoManuale;
      L     1;
      -I;
      T     "DatiOP170B".NumeroComandoManuale;
_003: NOP   0;
      A     L 1.0;
      A(;
      L     "DatiOP170B".NumeroComandoManuale;
      L     1;
      <I;
      );
      JNB   _004;
      L     10;
      T     "DatiOP170B".NumeroComandoManuale;
_004: NOP   0;
NETWORK
TITLE = UP\DOWN Table locker cylinder
      A     "On";
      =     L 1.0;
      A     L 1.0;
      A     "M11.2";
      A(;
      L     "DatiOP170B".NumeroComandoManuale;
      L     10;
      ==I;
      );
      A     "M16.7";
      AN    "REVERSE_TABLE_ROTATION";
      AN    "FWD_TABLE_ROTATION";
      =     L 1.1;
      A     L 1.1;
      A     "M22.4";
      AN    "M31.3";
      AN    "M32.5";
      S     "M32.5";
      R     "M32.4";
      A     L 1.1;
      A     "M22.5";
      AN    "M31.2";
      AN    "M32.4";
      S     "M32.4";
      R     "M32.5";
      A     L 1.1;
      BLD   102;
      =     "DatiOP170B".SegnalazioniServizio.TEXT10;
      A     L 1.0;
      A     "M22.0";
      R     "M32.5";
      A     L 1.0;
      A     "M22.1";
      R     "M32.4";
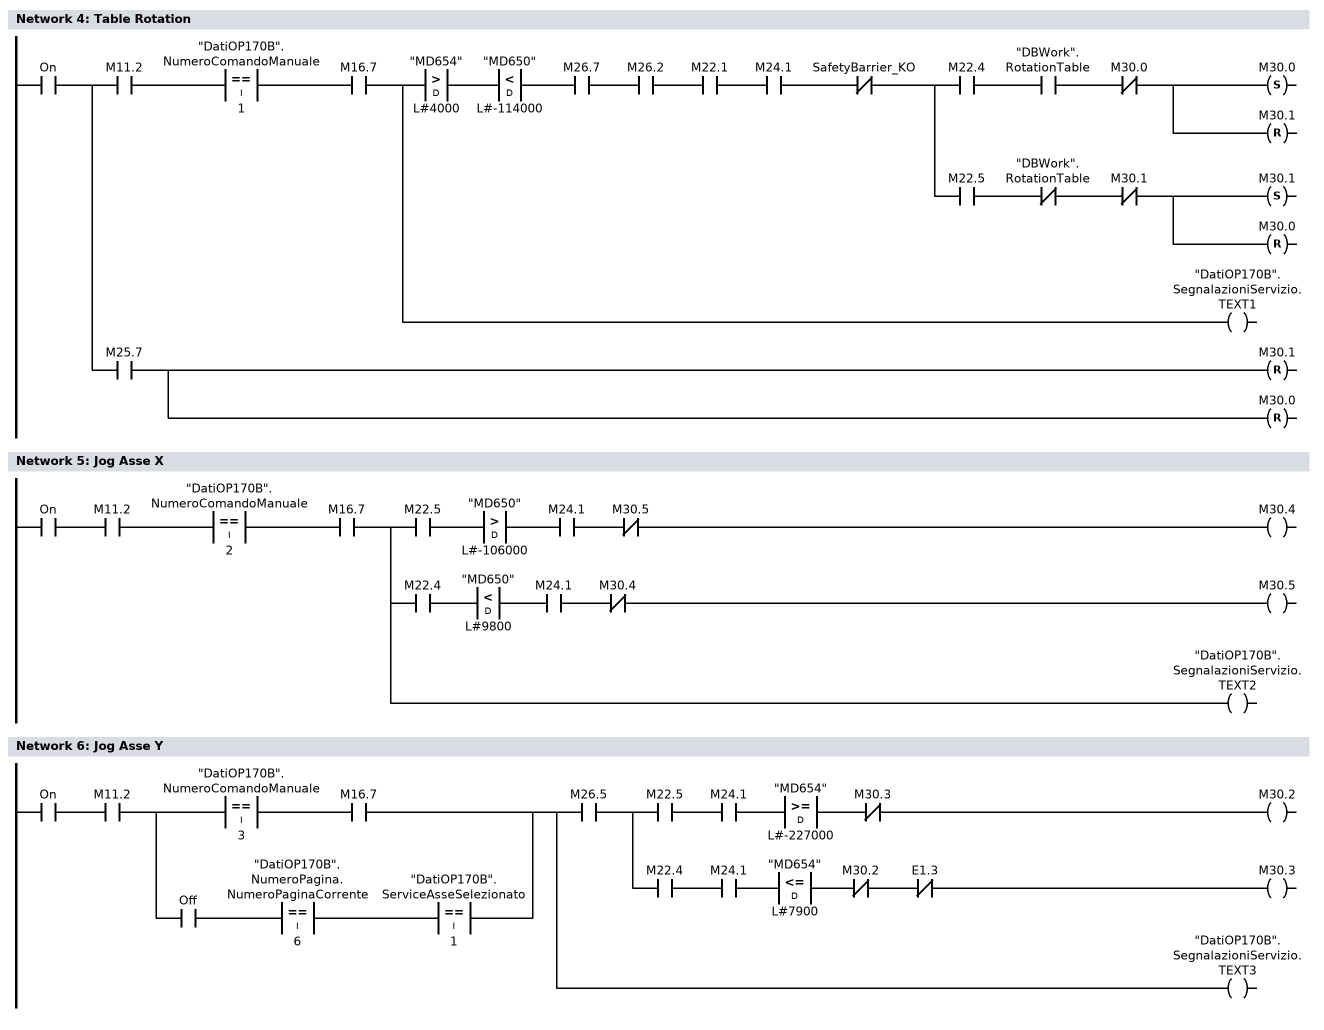
NETWORK
TITLE = Table Rotation
      A     "On";
      =     L 1.0;
      A     L 1.0;
      A     "M11.2";
      A(;
      L     "DatiOP170B".NumeroComandoManuale;
      L     1;
      ==I;
      );
      A     "M16.7";
      =     L 1.1;
      A     L 1.1;
      A(;
      L     "MD654";
      L     L#4000;
      >D;
      );
      A(;
      L     "MD650";
      L     L#-114000;
      <D;
      );
      A     "M26.7";
      A     "M26.2";
      A     "M22.1";
      A     "M24.1";
      AN    "SafetyBarrier_KO";
      =     L 1.2;
      A     L 1.2;
      A     "M22.4";
      A     "DBWork".RotationTable;
      AN    "M30.0";
      S     "M30.0";
      R     "M30.1";
      A     L 1.2;
      A     "M22.5";
      AN    "DBWork".RotationTable;
      AN    "M30.1";
      S     "M30.1";
      R     "M30.0";
      A     L 1.1;
      BLD   102;
      =     "DatiOP170B".SegnalazioniServizio.TEXT1;
      A     L 1.0;
      A     "M25.7";
      R     "M30.1";
      R     "M30.0";
NETWORK
TITLE = Jog Asse X
      A     "On";
      A     "M11.2";
      A(;
      A(;
      L     "DatiOP170B".NumeroComandoManuale;
      L     2;
      ==I;
      );
      A     "M16.7";
//     O     
//      U     "Off"
//      U(    
//      L     "DatiOP170B".NumeroPagina.NumeroPaginaCorrente
//      L     6
//      ==I   
//      )     
//      U(    
//      L     "DatiOP170B".ServiceAsseSelezionato
//      L     0
//      ==I   
//      )     
      );
      =     L 0.0;
      A     L 0.0;
      A     "M22.5";
      A(;
      L     "MD650";
      L     L#-106000;
      >D;
      );
      A     "M24.1";
      AN    "M30.5";
      =     "M30.4";
      A     L 0.0;
      A     "M22.4";
      A(;
      L     "MD650";
      L     L#9800;
      <D;
      );
      A     "M24.1";
      AN    "M30.4";
      =     "M30.5";
      A     L 0.0;
      BLD   102;
      =     "DatiOP170B".SegnalazioniServizio.TEXT2;
NETWORK
TITLE = Jog Asse Y
      A     "On";
      A     "M11.2";
      A(;
      A(;
      L     "DatiOP170B".NumeroComandoManuale;
      L     3;
      ==I;
      );
      A     "M16.7";
      O;
      A     "Off";
      A(;
      L     "DatiOP170B".NumeroPagina.NumeroPaginaCorrente;
      L     6;
      ==I;
      );
      A(;
      L     "DatiOP170B".ServiceAsseSelezionato;
      L     1;
      ==I;
      );
      );
      =     L 0.0;
      A     L 0.0;
      A     "M26.5";
      =     L 0.1;
      A     L 0.1;
      A     "M22.5";
      A     "M24.1";
      A(;
      L     "MD654";
      L     L#-227000;
      >=D;
      );
      AN    "M30.3";
      =     "M30.2";
      A     L 0.1;
      A     "M22.4";
      A     "M24.1";
      A(;
      L     "MD654";
      L     L#7900;
      <=D;
      );
      AN    "M30.2";
      AN    "E1.3";
      =     "M30.3";
      A     L 0.0;
      BLD   102;
      =     "DatiOP170B".SegnalazioniServizio.TEXT3;
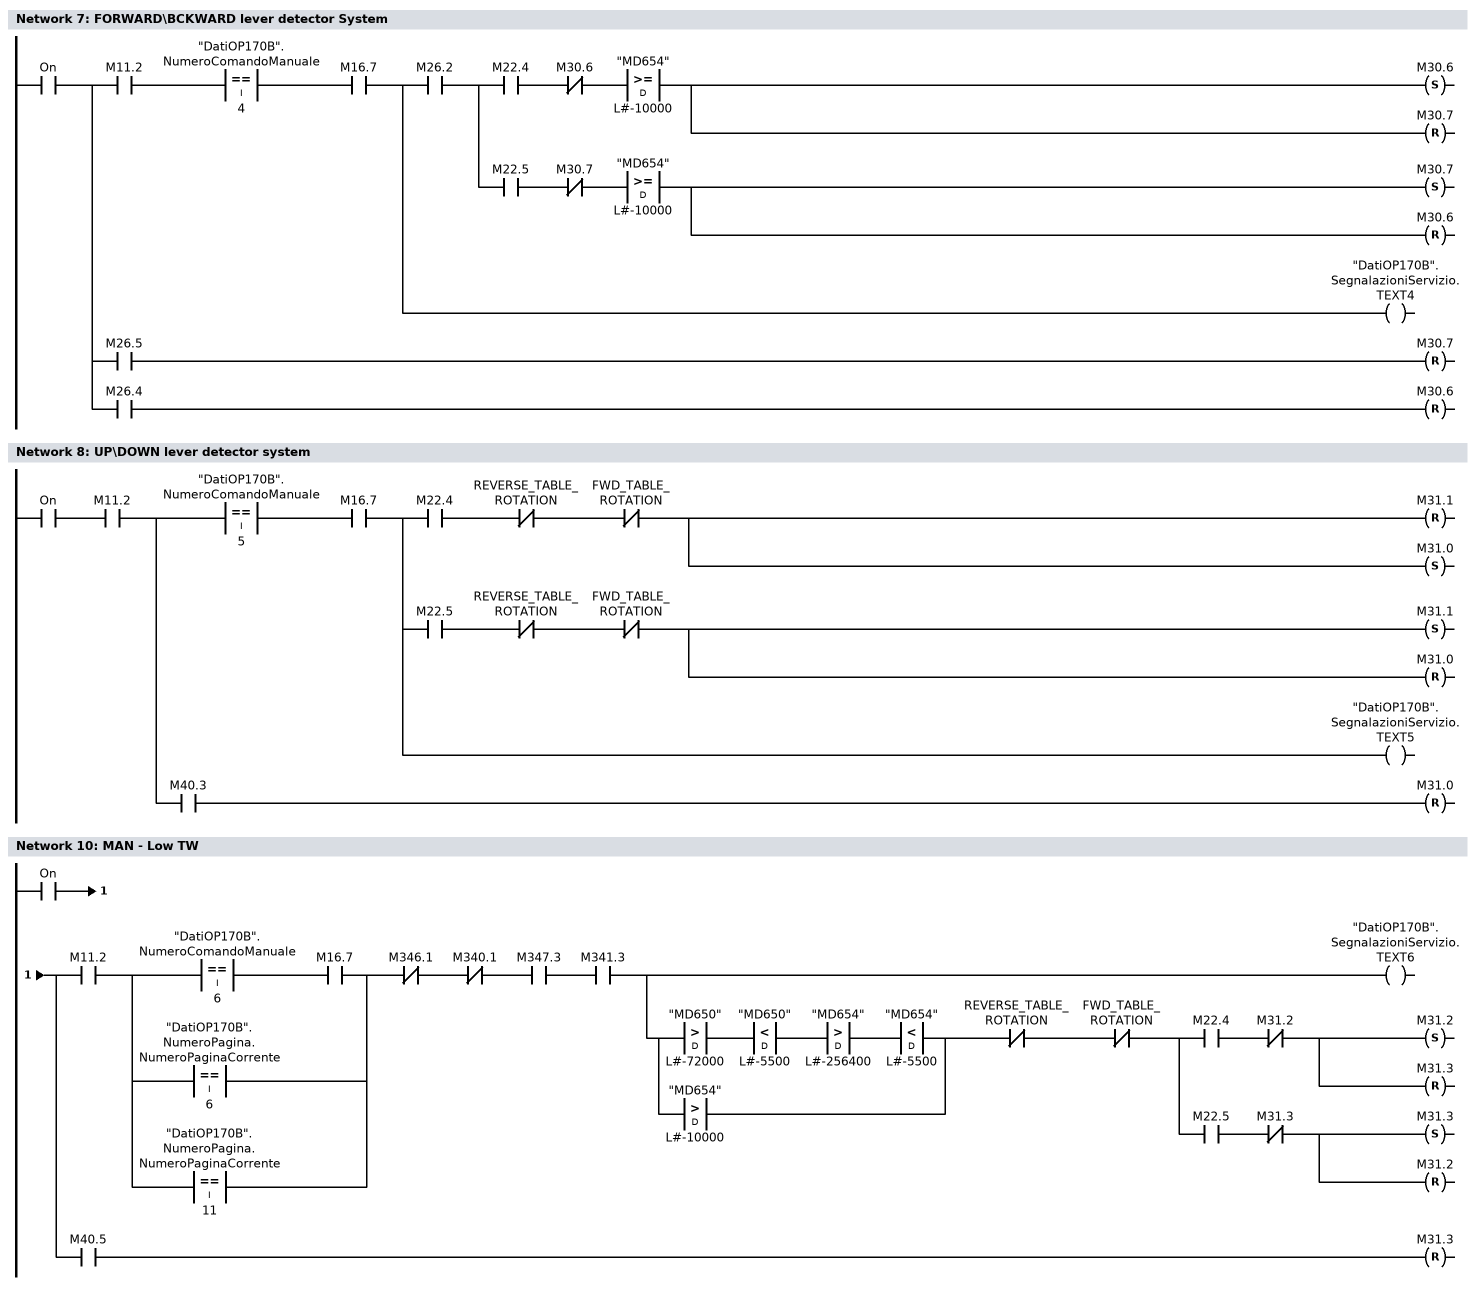
NETWORK
TITLE = FORWARD\BCKWARD lever detector System
//controllo fuori ingombro asse Y
      A     "On";
      =     L 1.0;
      A     L 1.0;
      A     "M11.2";
      A(;
      L     "DatiOP170B".NumeroComandoManuale;
      L     4;
      ==I;
      );
      A     "M16.7";
      =     L 1.1;
      A     L 1.1;
      A     "M26.2";
      =     L 1.2;
      A     L 1.2;
      A     "M22.4";
      AN    "M30.6";
      A(;
      L     "MD654";
      L     L#-10000;
      >=D;
      );
      S     "M30.6";
      R     "M30.7";
      A     L 1.2;
      A     "M22.5";
      AN    "M30.7";
      A(;
      L     "MD654";
      L     L#-10000;
      >=D;
      );
      S     "M30.7";
      R     "M30.6";
      A     L 1.1;
      BLD   102;
      =     "DatiOP170B".SegnalazioniServizio.TEXT4;
      A     L 1.0;
      A     "M26.5";
      R     "M30.7";
      A     L 1.0;
      A     "M26.4";
      R     "M30.6";
NETWORK
TITLE = UP\DOWN lever detector system
      A     "On";
      A     "M11.2";
      =     L 1.0;
      A     L 1.0;
      A(;
      L     "DatiOP170B".NumeroComandoManuale;
      L     5;
      ==I;
      );
      A     "M16.7";
      =     L 1.1;
      A     L 1.1;
      A     "M22.4";
      AN    "REVERSE_TABLE_ROTATION";
      AN    "FWD_TABLE_ROTATION";
      R     "M31.1";
      S     "M31.0";
      A     L 1.1;
      A     "M22.5";
      AN    "REVERSE_TABLE_ROTATION";
      AN    "FWD_TABLE_ROTATION";
      S     "M31.1";
      R     "M31.0";
      A     L 1.1;
      BLD   102;
      =     "DatiOP170B".SegnalazioniServizio.TEXT5;
      A     L 1.0;
      A     "M40.3";
      R     "M31.0";
NETWORK
TITLE = UP\DOWN Torch Welding Machine
//      U     "On"
//      =     L      0.0
//      U     L      0.0
//      U     "M11.2"
//      U(    
//      U(    
//      L     "DatiOP170B".NumeroComandoManuale
//      L     6
//      ==I   
//      )     
//      U     "M16.7"
//      O     
//      U(    
//      O(    
//      L     "DatiOP170B".NumeroPagina.NumeroPaginaCorrente
//      L     6
//      ==I   
//      )     
//      O(    
//      L     "DatiOP170B".NumeroPagina.NumeroPaginaCorrente
//      L     11
//      ==I   
//      )     
//      )     
//      UN    "M346.1"
//      UN    "M340.1"
//      U     "M347.3"
//      U     "M341.3"
//      )     
//      =     L      0.1
//      U     L      0.1
//      U(    
//      U(    
//      L     "MD650"
//      L     L#-72000
//      >D    
//      )     
//      U(    
//      L     "MD650"
//      L     L#-5500
//      <D    
//      )     
//      U(    
//      L     "MD654"
//      L     L#-256400
//      >D    
//      )     
//      U(    
//      L     "MD654"
//      L     L#-5500
//      <D    
//      )     
//      O(    
//      L     "MD654"
//      L     -10000
//      >D    
//      )     
//      )     
//      UN    "REVERSE_TABLE_ROTATION"
//      UN    "FWD_TABLE_ROTATION"
//      =     L      0.2
//      U     L      0.2
//      U     "M22.4"
//      UN    "M31.2"
//      S     "M31.2"
//      R     "M31.3"
//      U     L      0.2
//      U     "M22.5"
//      UN    "M31.3"
//      S     "M31.3"
//      R     "M31.2"
//      U     L      0.1
//      BLD   102
//      =     "DatiOP170B".SegnalazioniServizio.TEXT6
//      U     L      0.0
//      U     "M40.5"
//      R     "M31.3"
//  A     L      0.0
// A     "M24.1"
// R     "M31.2"
NETWORK
TITLE = MAN - Low TW
      A     "On";
      =     L 1.0;
      A     L 1.0;
      A     "M11.2";
      A(;
      A(;
      L     "DatiOP170B".NumeroComandoManuale;
      L     6;
      ==I;
      );
      A     "M16.7";
      O(;
      L     "DatiOP170B".NumeroPagina.NumeroPaginaCorrente;
      L     6;
      ==I;
      );
      O(;
      L     "DatiOP170B".NumeroPagina.NumeroPaginaCorrente;
      L     11;
      ==I;
      );
      );
      AN    "M346.1";
      AN    "M340.1";
      A     "M347.3";
      A     "M341.3";
      =     L 1.1;
      A     L 1.1;
      BLD   102;
      =     "DatiOP170B".SegnalazioniServizio.TEXT6;
      A     L 1.1;
      A(;
      A(;
      L     "MD650";
      L     L#-72000;
      >D;
      );
      A(;
      L     "MD650";
      L     L#-5500;
      <D;
      );
      A(;
      L     "MD654";
      L     L#-256400;
      >D;
      );
      A(;
      L     "MD654";
      L     L#-5500;
      <D;
      );
      O(;
      L     "MD654";
      L     L#-10000;
      >D;
      );
      );
      AN    "REVERSE_TABLE_ROTATION";
      AN    "FWD_TABLE_ROTATION";
      =     L 1.2;
      A     L 1.2;
      A     "M22.4";
      AN    "M31.2";
      S     "M31.2";
      R     "M31.3";
      A     L 1.2;
      A     "M22.5";
      AN    "M31.3";
      S     "M31.3";
      R     "M31.2";
      A     L 1.0;
      A     "M40.5";
      R     "M31.3";
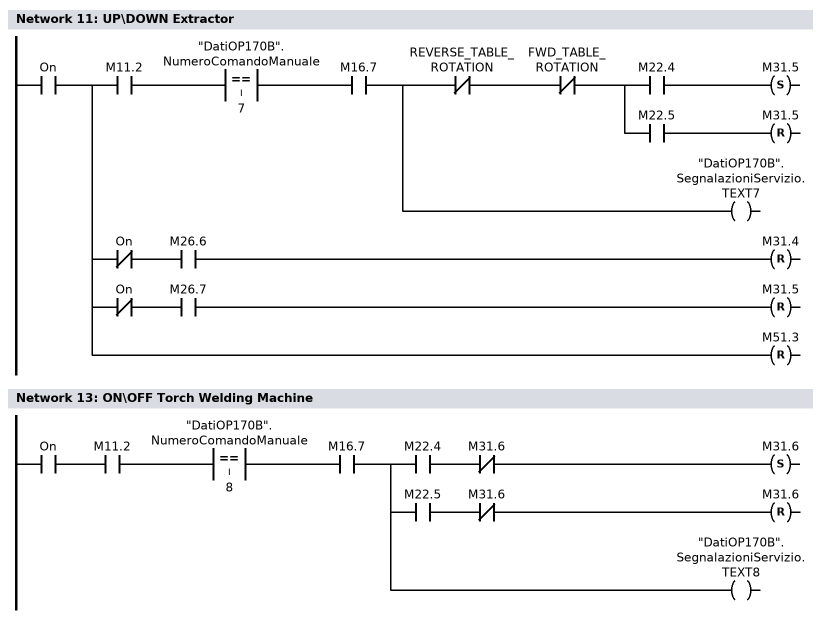
NETWORK
TITLE = UP\DOWN Extractor
      A     "On";
      =     L 1.0;
      A     L 1.0;
      A     "M11.2";
      A(;
      L     "DatiOP170B".NumeroComandoManuale;
      L     7;
      ==I;
      );
      A     "M16.7";
      =     L 1.1;
      A     L 1.1;
      AN    "REVERSE_TABLE_ROTATION";
      AN    "FWD_TABLE_ROTATION";
      =     L 1.2;
      A     L 1.2;
      A     "M22.4";
      S     "M31.5";
      A     L 1.2;
      A     "M22.5";
      R     "M31.5";
      A     L 1.1;
      BLD   102;
      =     "DatiOP170B".SegnalazioniServizio.TEXT7;
      A     L 1.0;
      AN    "On";
      A     "M26.6";
      R     "M31.4";
      A     L 1.0;
      AN    "On";
      A     "M26.7";
      R     "M31.5";
      A     L 1.0;
      BLD   102;
      R     "M51.3";
NETWORK
TITLE =
NETWORK
TITLE = ON\OFF Torch Welding Machine
      A     "On";
      A     "M11.2";
      A(;
      L     "DatiOP170B".NumeroComandoManuale;
      L     8;
      ==I;
      );
      A     "M16.7";
      =     L 1.0;
      A     L 1.0;
      A     "M22.4";
      AN    "M31.6";
      S     "M31.6";
      A     L 1.0;
      A     "M22.5";
      AN    "M31.6";
      R     "M31.6";
      A     L 1.0;
      BLD   102;
      =     "DatiOP170B".SegnalazioniServizio.TEXT8;
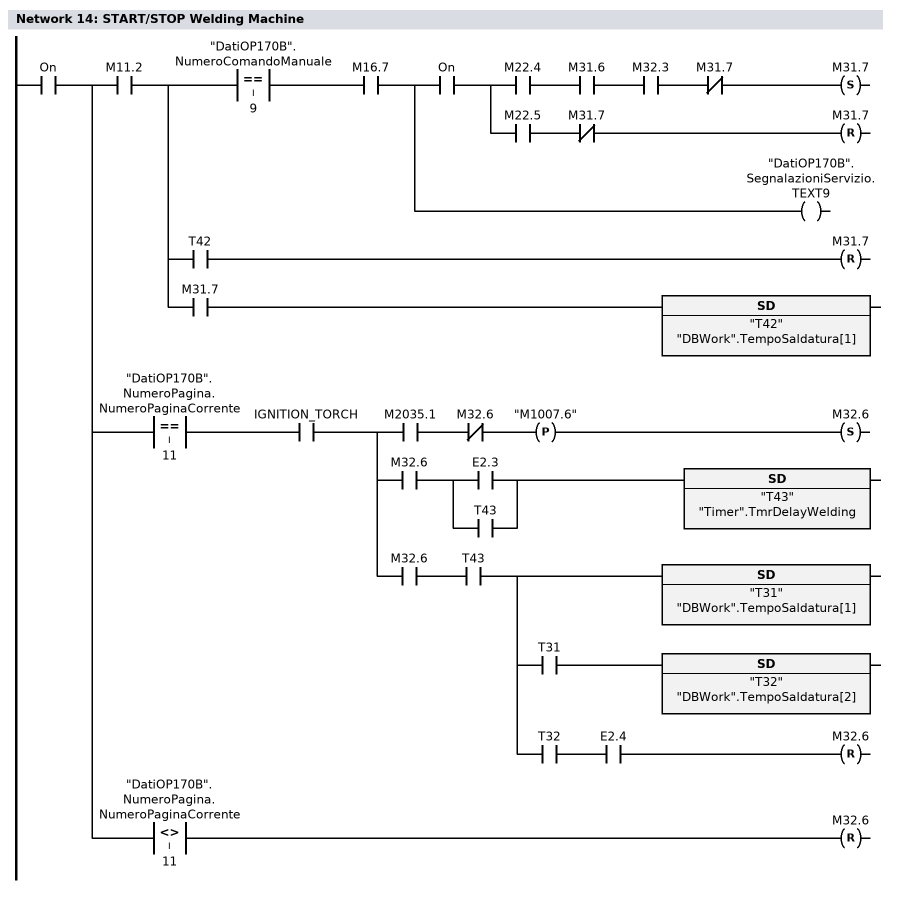
NETWORK
TITLE = START/STOP Welding Machine
      A     "On";
      =     L 1.0;
      A     L 1.0;
      A     "M11.2";
      =     L 1.1;
      A     L 1.1;
      A(;
      L     "DatiOP170B".NumeroComandoManuale;
      L     9;
      ==I;
      );
      A     "M16.7";
      =     L 1.2;
      A     L 1.2;
      A     "On";
      =     L 1.3;
      A     L 1.3;
      A     "M22.4";
      A     "M31.6";
      A     "M32.3";
      AN    "M31.7";
      S     "M31.7";
      A     L 1.3;
      A     "M22.5";
      AN    "M31.7";
      R     "M31.7";
      A     L 1.2;
      BLD   102;
      =     "DatiOP170B".SegnalazioniServizio.TEXT9;
      A     L 1.1;
      A     "T42";
      R     "M31.7";
      A     L 1.1;
      A     "M31.7";
      L     "DBWork".TempoSaldatura[1];
      SD    "T42";
      A     L 1.0;
      A(;
      L     "DatiOP170B".NumeroPagina.NumeroPaginaCorrente;
      L     11;
      ==I;
      );
      A     "IGNITION_TORCH";
      =     L 1.1;
      A     L 1.1;
      A     "M2035.1";
      AN    "M32.6";
      FP    "M1007.6";
      S     "M32.6";
      A     L 1.1;
      A     "M32.6";
      A(;
      O     "E2.3";
      O     "T43";
      );
      L     "Timer".TmrDelayWelding;
      SD    "T43";
      A     L 1.1;
      A     "M32.6";
      A     "T43";
      =     L 1.2;
      A     L 1.2;
      BLD   102;
      L     "DBWork".TempoSaldatura[1];
      SD    "T31";
      A     L 1.2;
      A     "T31";
      L     "DBWork".TempoSaldatura[2];
      SD    "T32";
      A     L 1.2;
      A     "T32";
      A     "E2.4";
      R     "M32.6";
      A     L 1.0;
      A(;
      L     "DatiOP170B".NumeroPagina.NumeroPaginaCorrente;
      L     11;
      <>I;
      );
      R     "M32.6";
END_FUNCTION

FUNCTION "FC14 - AUTOMATIC" : VOID	// FC 14
TITLE = Automatic cycle management
VERSION : 0.1
VAR_TEMP
  MinX : DINT ;
  MinY : DINT ;
  MaxX : DINT ;
  MaxY : DINT ;
END_VAR
BEGIN
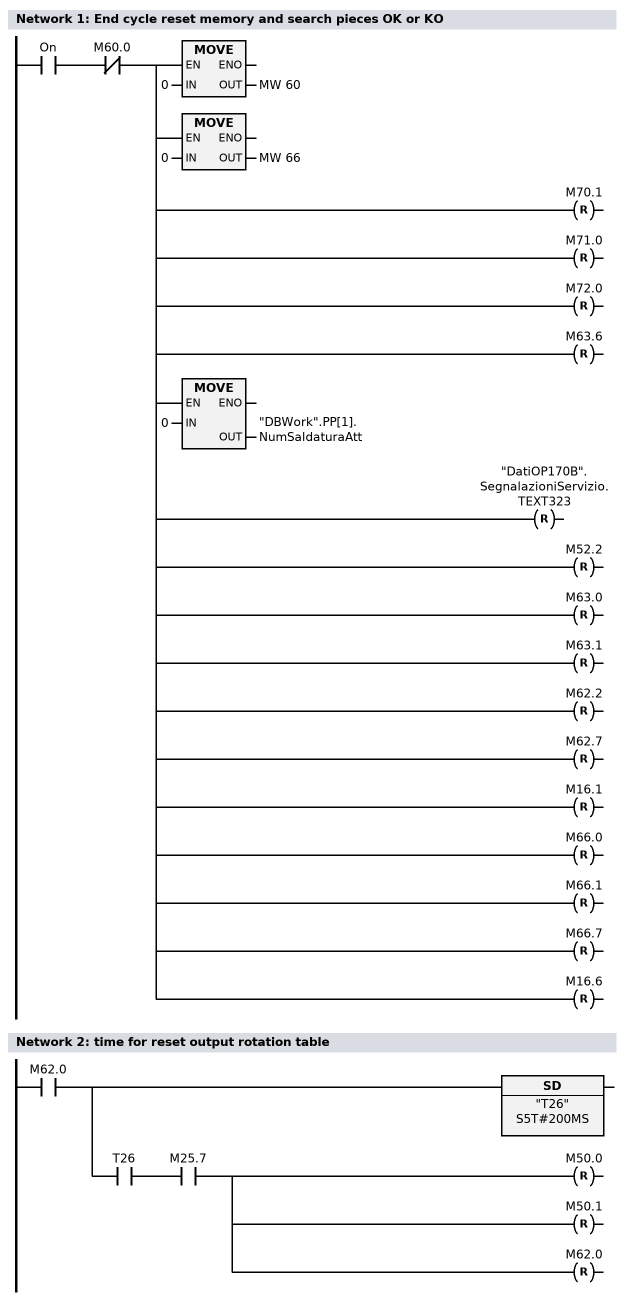
NETWORK
TITLE = End cycle reset memory and search pieces OK or KO
      A     "On";
      AN    "M60.0";
      =     L 16.0;
      A     L 16.0;
      JNB   _001;
      L     0;
      T     MW 60;
_001: NOP   0;
      A     L 16.0;
      JNB   _002;
      L     0;
      T     MW 66;
_002: NOP   0;
      A     L 16.0;
      BLD   102;
      R     "M70.1";
      A     L 16.0;
      BLD   102;
      R     "M71.0";
      A     L 16.0;
      BLD   102;
      R     "M72.0";
      A     L 16.0;
      BLD   102;
      R     "M63.6";
      A     L 16.0;
      JNB   _003;
      L     0;
      T     "DBWork".PP[1].NumSaldaturaAtt;
_003: NOP   0;
      A     L 16.0;
      BLD   102;
      R     "DatiOP170B".SegnalazioniServizio.TEXT323;
      A     L 16.0;
      BLD   102;
      R     "M52.2";
      A     L 16.0;
      BLD   102;
      R     "M63.0";
      A     L 16.0;
      BLD   102;
      R     "M63.1";
      A     L 16.0;
      BLD   102;
      R     "M62.2";
      A     L 16.0;
      BLD   102;
      R     "M62.7";
      A     L 16.0;
      BLD   102;
      R     "M16.1";
      A     L 16.0;
      BLD   102;
      R     "M66.0";
      A     L 16.0;
      BLD   102;
      R     "M66.1";
      A     L 16.0;
      BLD   102;
      R     "M66.7";
      A     L 16.0;
      BLD   102;
      R     "M16.6";
NETWORK
TITLE = time for reset output rotation table
//Reset Output Rotation Table 
      A     "M62.0";
      =     L 16.0;
      A     L 16.0;
      BLD   102;
      L     S5T#200MS;
      SD    "T26";
      A     L 16.0;
      A     "T26";
      A     "M25.7";
      R     "M50.0";
      R     "M50.1";
      R     "M62.0";
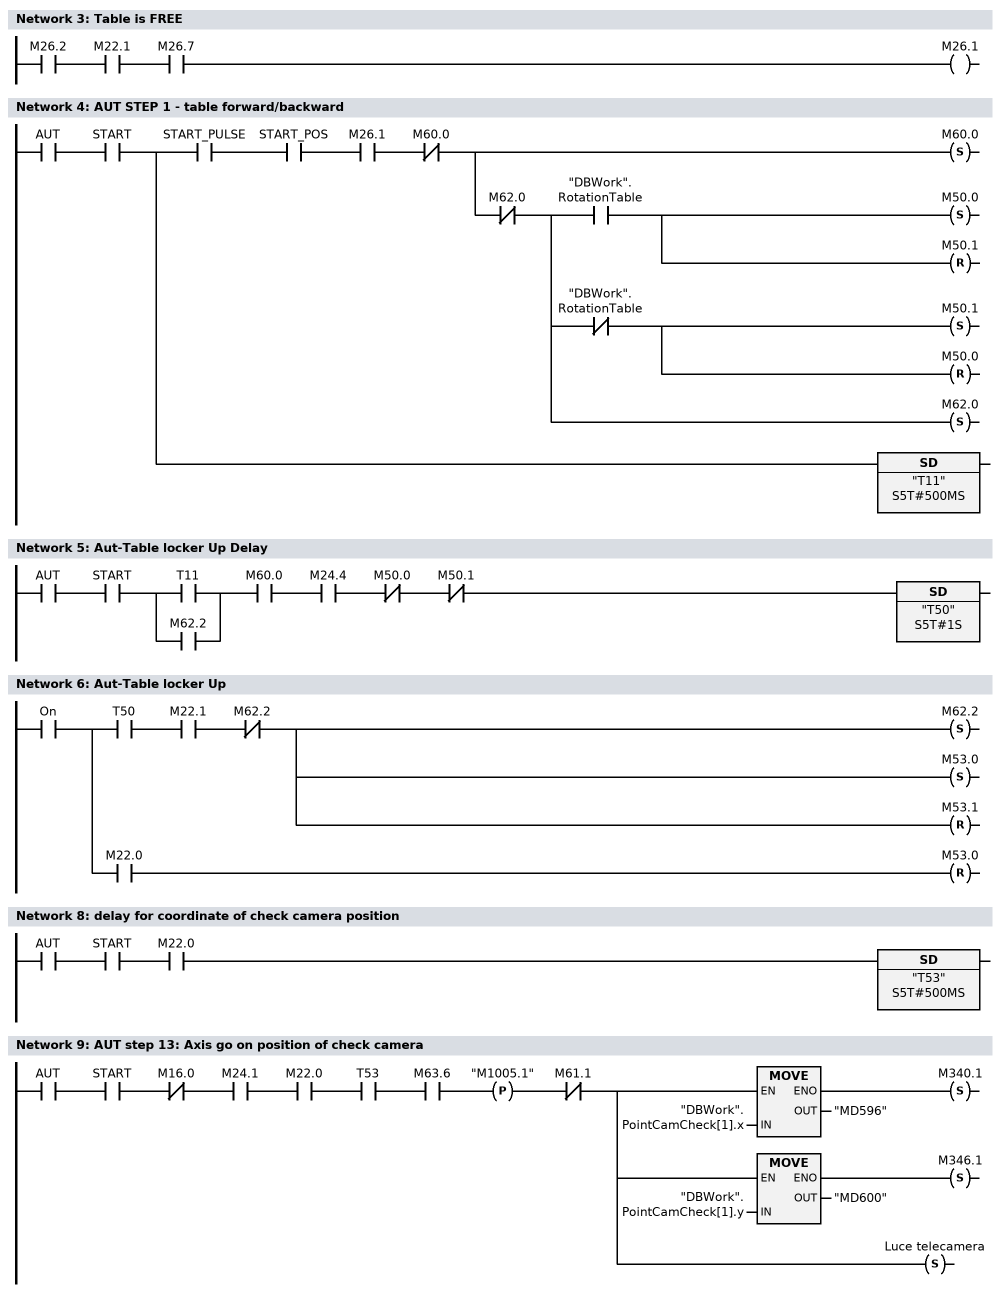
NETWORK
TITLE = Table is FREE
      A     "M26.2";
      A     "M22.1";
      A     "M26.7";
      =     "M26.1";
NETWORK
TITLE = AUT STEP 1 - table forward/backward
      A     "AUT";
      A     "START";
      =     L 16.0;
      A     L 16.0;
      A     "START_PULSE";
      A     "START_POS";
      A     "M26.1";
      AN    "M60.0";
      =     L 16.1;
      A     L 16.1;
      BLD   102;
      S     "M60.0";
      A     L 16.1;
      AN    "M62.0";
      =     L 16.2;
      A     L 16.2;
      A     "DBWork".RotationTable;
      S     "M50.0";
      R     "M50.1";
      A     L 16.2;
      AN    "DBWork".RotationTable;
      S     "M50.1";
      R     "M50.0";
      A     L 16.2;
      BLD   102;
      S     "M62.0";
      A     L 16.0;
      BLD   102;
      L     S5T#500MS;
      SD    "T11";
NETWORK
TITLE = Aut-Table locker Up Delay
      A     "AUT";
      A     "START";
      A(;
      O     "T11";
      O     "M62.2";
      );
      A     "M60.0";
      A     "M24.4";
      AN    "M50.0";
      AN    "M50.1";
      L     S5T#1S;
      SD    "T50";
NETWORK
TITLE = Aut-Table locker Up
      A     "On";
      =     L 16.0;
      A     L 16.0;
      A     "T50";
      A     "M22.1";
      AN    "M62.2";
      S     "M62.2";
      S     "M53.0";
      R     "M53.1";
      A     L 16.0;
      A     "M22.0";
      R     "M53.0";
NETWORK
TITLE = Check With OMRON if Component is OK
NETWORK
TITLE = delay for coordinate of check camera position
      A     "AUT";
      A     "START";
      A     "M22.0";
      L     S5T#500MS;
      SD    "T53";
NETWORK
TITLE = AUT step 13: Axis go on position of check camera
      A     "AUT";
      A     "START";
      AN    "M16.0";
      A     "M24.1";
      A     "M22.0";
      A     "T53";
      A     "M63.6";
      FP    "M1005.1";
      AN    "M61.1";
      =     L 16.0;
      A     L 16.0;
      JNB   _004;
      L     "DBWork".PointCamCheck[1].x;
      T     "MD596";
      SET;
      SAVE;
      CLR;
_004: A     BR;
      S     "M340.1";
      A     L 16.0;
      JNB   _005;
      L     "DBWork".PointCamCheck[1].y;
      T     "MD600";
      SET;
      SAVE;
      CLR;
_005: A     BR;
      S     "M346.1";
      A     L 16.0;
      BLD   102;
      S     "Luce telecamera";
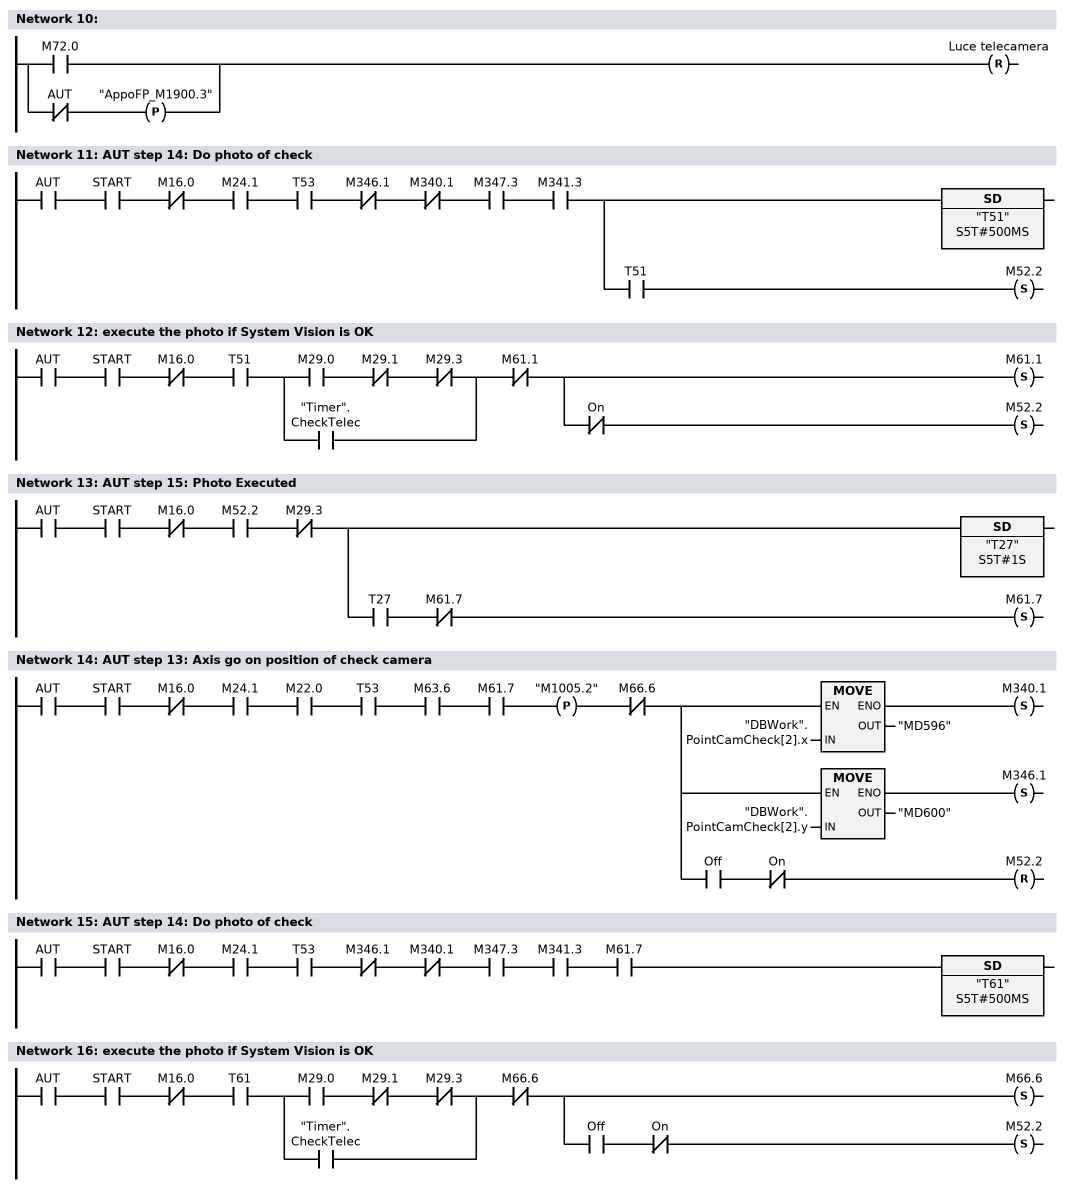
NETWORK
TITLE =
      O     "M72.0";
      O(;
      AN    "AUT";
      FP    "AppoFP_M1900.3";
      );
      R     "Luce telecamera";
NETWORK
TITLE = AUT step 14: Do photo of check 
      A     "AUT";
      A     "START";
      AN    "M16.0";
      A     "M24.1";
      A     "T53";
      AN    "M346.1";
      AN    "M340.1";
      A     "M347.3";
      A     "M341.3";
      =     L 16.0;
      A     L 16.0;
      BLD   102;
      L     S5T#500MS;
      SD    "T51";
      A     L 16.0;
      A     "T51";
      S     "M52.2";
NETWORK
TITLE = execute the photo if System Vision is OK
      A     "AUT";
      A     "START";
      AN    "M16.0";
      A     "T51";
      A(;
      A     "M29.0";
      AN    "M29.1";
      AN    "M29.3";
      O     "Timer".CheckTelec;
      );
      AN    "M61.1";
      =     L 16.0;
      A     L 16.0;
      BLD   102;
      S     "M61.1";
      A     L 16.0;
      AN    "On";
      S     "M52.2";
NETWORK
TITLE = AUT step 15: Photo Executed
      A     "AUT";
      A     "START";
      AN    "M16.0";
      A     "M52.2";
      AN    "M29.3";
      =     L 16.0;
      A     L 16.0;
      BLD   102;
      L     S5T#1S;
      SD    "T27";
      A     L 16.0;
      A     "T27";
      AN    "M61.7";
      S     "M61.7";
NETWORK
TITLE = AUT step 13: Axis go on position of check camera
      A     "AUT";
      A     "START";
      AN    "M16.0";
      A     "M24.1";
      A     "M22.0";
      A     "T53";
      A     "M63.6";
      A     "M61.7";
      FP    "M1005.2";
      AN    "M66.6";
      =     L 16.0;
      A     L 16.0;
      JNB   _006;
      L     "DBWork".PointCamCheck[2].x;
      T     "MD596";
      SET;
      SAVE;
      CLR;
_006: A     BR;
      S     "M340.1";
      A     L 16.0;
      JNB   _007;
      L     "DBWork".PointCamCheck[2].y;
      T     "MD600";
      SET;
      SAVE;
      CLR;
_007: A     BR;
      S     "M346.1";
      A     L 16.0;
      A     "Off";
      AN    "On";
      R     "M52.2";
NETWORK
TITLE = AUT step 14: Do photo of check 
      A     "AUT";
      A     "START";
      AN    "M16.0";
      A     "M24.1";
      A     "T53";
      AN    "M346.1";
      AN    "M340.1";
      A     "M347.3";
      A     "M341.3";
      A     "M61.7";
      L     S5T#500MS;
      SD    "T61";
NETWORK
TITLE = execute the photo if System Vision is OK
      A     "AUT";
      A     "START";
      AN    "M16.0";
      A     "T61";
      A(;
      A     "M29.0";
      AN    "M29.1";
      AN    "M29.3";
      O     "Timer".CheckTelec;
      );
      AN    "M66.6";
      =     L 16.0;
      A     L 16.0;
      BLD   102;
      S     "M66.6";
      A     L 16.0;
      A     "Off";
      AN    "On";
      S     "M52.2";
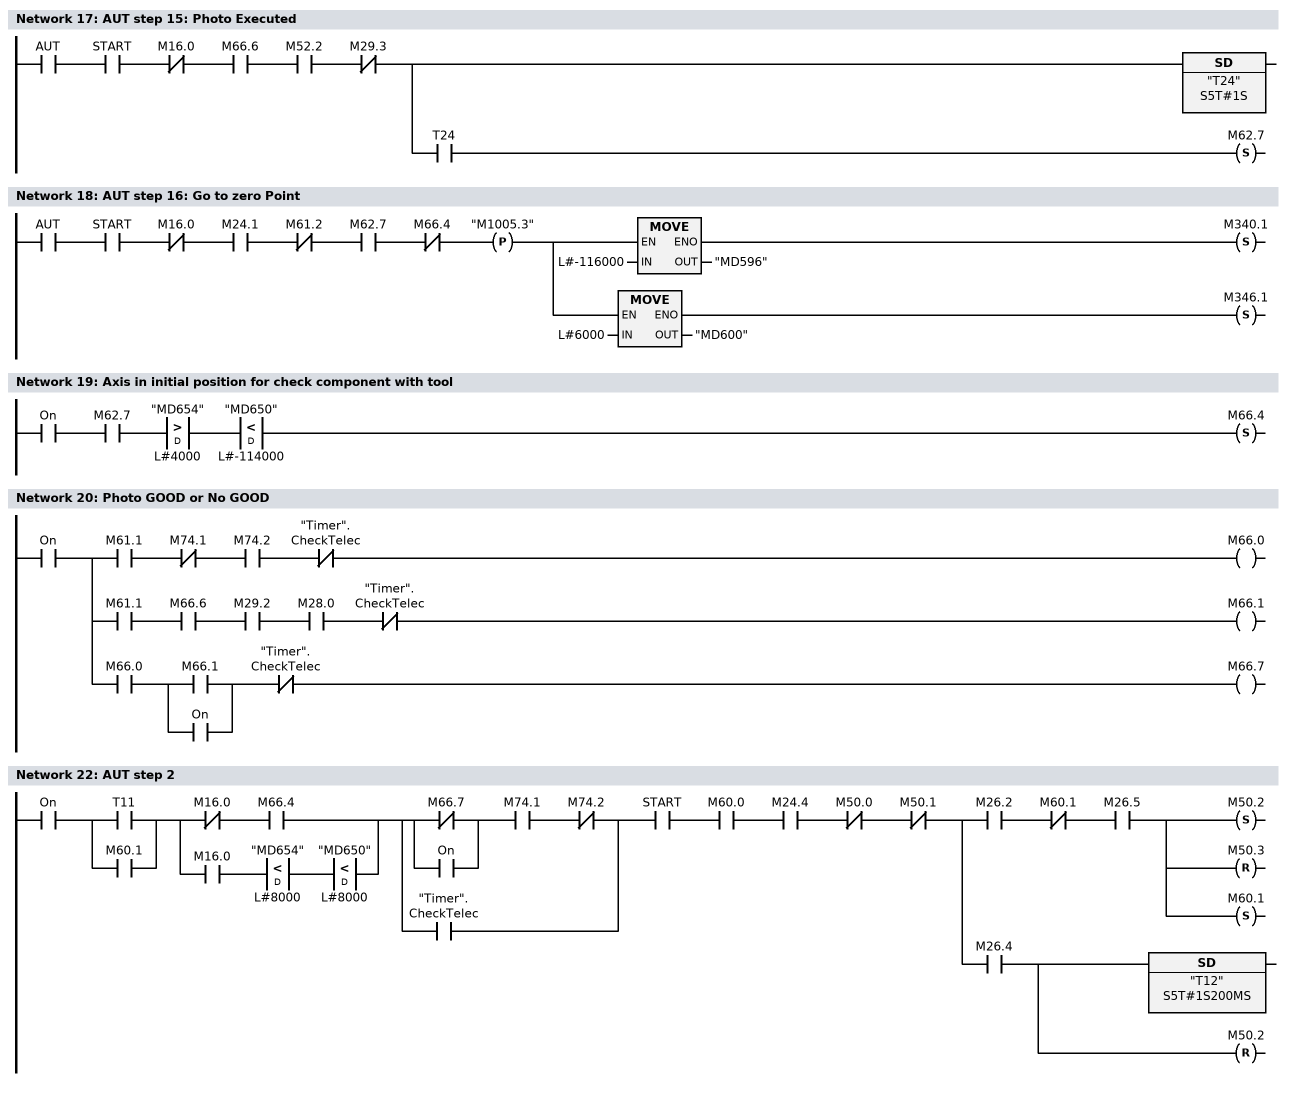
NETWORK
TITLE = AUT step 15: Photo Executed
      A     "AUT";
      A     "START";
      AN    "M16.0";
      A     "M66.6";
      A     "M52.2";
      AN    "M29.3";
      =     L 16.0;
      A     L 16.0;
      BLD   102;
      L     S5T#1S;
      SD    "T24";
      A     L 16.0;
      A     "T24";
      S     "M62.7";
NETWORK
TITLE = AUT step 16: Go to zero Point
      A     "AUT";
      A     "START";
      AN    "M16.0";
      A     "M24.1";
      AN    "M61.2";
      A     "M62.7";
      AN    "M66.4";
      FP    "M1005.3";
      =     L 16.0;
      A     L 16.0;
      JNB   _008;
      L     L#-116000;
      T     "MD596";
      SET;
      SAVE;
      CLR;
_008: A     BR;
      S     "M340.1";
      A     L 16.0;
      JNB   _009;
      L     L#6000;
      T     "MD600";
      SET;
      SAVE;
      CLR;
_009: A     BR;
      S     "M346.1";
NETWORK
TITLE = Axis in initial position for check component with tool
      A     "On";
      A     "M62.7";
      A(;
      L     "MD654";
      L     L#4000;
      >D;
      );
      A(;
      L     "MD650";
      L     L#-114000;
      <D;
      );
      S     "M66.4";
NETWORK
TITLE = Photo GOOD or No GOOD
      A     "On";
      =     L 16.0;
      A     L 16.0;
      A     "M61.1";
      AN    "M74.1";
      A     "M74.2";
      AN    "Timer".CheckTelec;
      =     "M66.0";
      A     L 16.0;
      A     "M61.1";
      A     "M66.6";
      A     "M29.2";
      A     "M28.0";
      AN    "Timer".CheckTelec;
      =     "M66.1";
      A     L 16.0;
      A     "M66.0";
      A(;
      O     "M66.1";
      O     "On";
      );
      AN    "Timer".CheckTelec;
      =     "M66.7";
NETWORK
TITLE =
NETWORK
TITLE = AUT step 2
//Step 2: System Detector Forward ed 
      A     "On";
      A(;
      O     "T11";
      O     "M60.1";
      );
      A(;
      AN    "M16.0";
      A     "M66.4";
      O;
      A     "M16.0";
      A(;
      L     "MD654";
      L     L#8000;
      <D;
      );
      A(;
      L     "MD650";
      L     L#8000;
      <D;
      );
      );
      A(;
      A(;
      ON    "M66.7";
      O     "On";
      );
      A     "M74.1";
      AN    "M74.2";
      O     "Timer".CheckTelec;
      );
      A     "START";
      A     "M60.0";
      A     "M24.4";
      AN    "M50.0";
      AN    "M50.1";
      =     L 16.0;
      A     L 16.0;
      A     "M26.2";
      AN    "M60.1";
      A     "M26.5";
      S     "M50.2";
      R     "M50.3";
      S     "M60.1";
      A     L 16.0;
      A     "M26.4";
      L     S5T#1S200MS;
      SD    "T12";
      R     "M50.2";
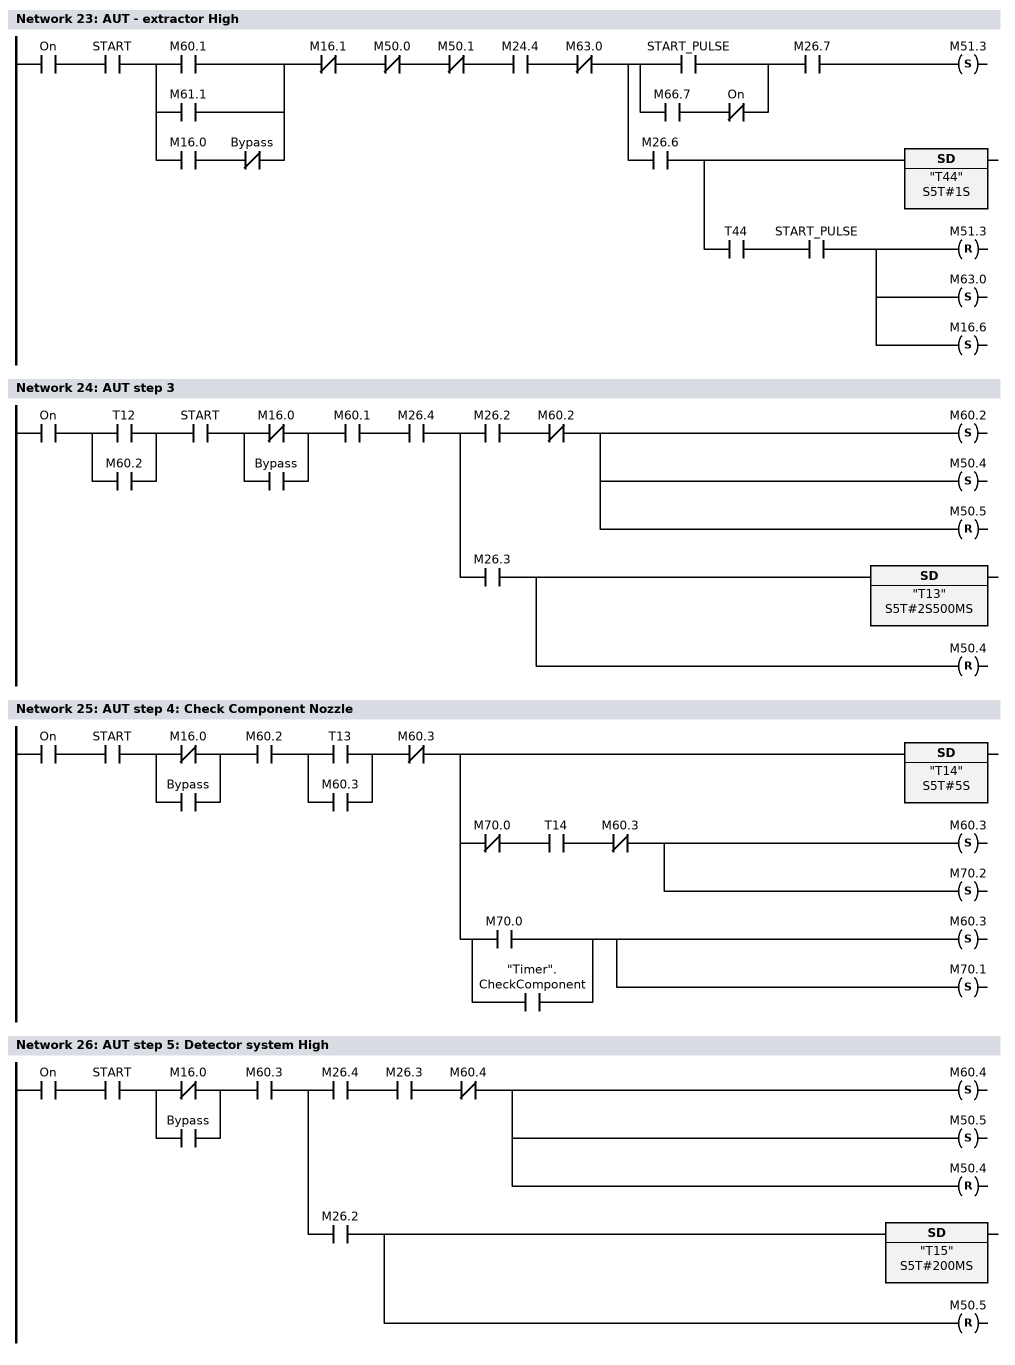
NETWORK
TITLE = AUT - extractor High
//Insert Extractor , extract worked pieces, i make it together Step 2
      A     "On";
      A     "START";
      A(;
      O     "M60.1";
      O     "M61.1";
      O;
      A     "M16.0";
      AN    "Bypass";
      );
      AN    "M16.1";
      AN    "M50.0";
      AN    "M50.1";
      A     "M24.4";
      AN    "M63.0";
      =     L 16.0;
      A     L 16.0;
      A(;
      O     "START_PULSE";
      O;
      A     "M66.7";
      AN    "On";
      );
      A     "M26.7";
      S     "M51.3";
      A     L 16.0;
      A     "M26.6";
      =     L 16.1;
      A     L 16.1;
      BLD   102;
      L     S5T#1S;
      SD    "T44";
      A     L 16.1;
      A     "T44";
      A     "START_PULSE";
      R     "M51.3";
      S     "M63.0";
      S     "M16.6";
NETWORK
TITLE = AUT step 3
//Step 3: System Detector Low
      A     "On";
      A(;
      O     "T12";
      O     "M60.2";
      );
      A     "START";
      A(;
      ON    "M16.0";
      O     "Bypass";
      );
      A     "M60.1";
      A     "M26.4";
      =     L 16.0;
      A     L 16.0;
      A     "M26.2";
      AN    "M60.2";
      S     "M60.2";
      S     "M50.4";
      R     "M50.5";
      A     L 16.0;
      A     "M26.3";
      L     S5T#2S500MS;
      SD    "T13";
      R     "M50.4";
NETWORK
TITLE = AUT step 4: Check Component Nozzle
//check if is possible work pieces
//
      A     "On";
      A     "START";
      A(;
      ON    "M16.0";
      O     "Bypass";
      );
      A     "M60.2";
      A(;
      O     "T13";
      O     "M60.3";
      );
      AN    "M60.3";
      =     L 16.0;
      A     L 16.0;
      BLD   102;
      L     S5T#5S;
      SD    "T14";
      A     L 16.0;
      AN    "M70.0";
      A     "T14";
      AN    "M60.3";
      S     "M60.3";
      S     "M70.2";
      A     L 16.0;
      A(;
      O     "M70.0";
      O     "Timer".CheckComponent;
      );
      S     "M60.3";
      S     "M70.1";
NETWORK
TITLE = AUT step 5: Detector system High
      A     "On";
      A     "START";
      A(;
      ON    "M16.0";
      O     "Bypass";
      );
      A     "M60.3";
      =     L 16.0;
      A     L 16.0;
      A     "M26.4";
      A     "M26.3";
      AN    "M60.4";
      S     "M60.4";
      S     "M50.5";
      R     "M50.4";
      A     L 16.0;
      A     "M26.2";
      L     S5T#200MS;
      SD    "T15";
      R     "M50.5";
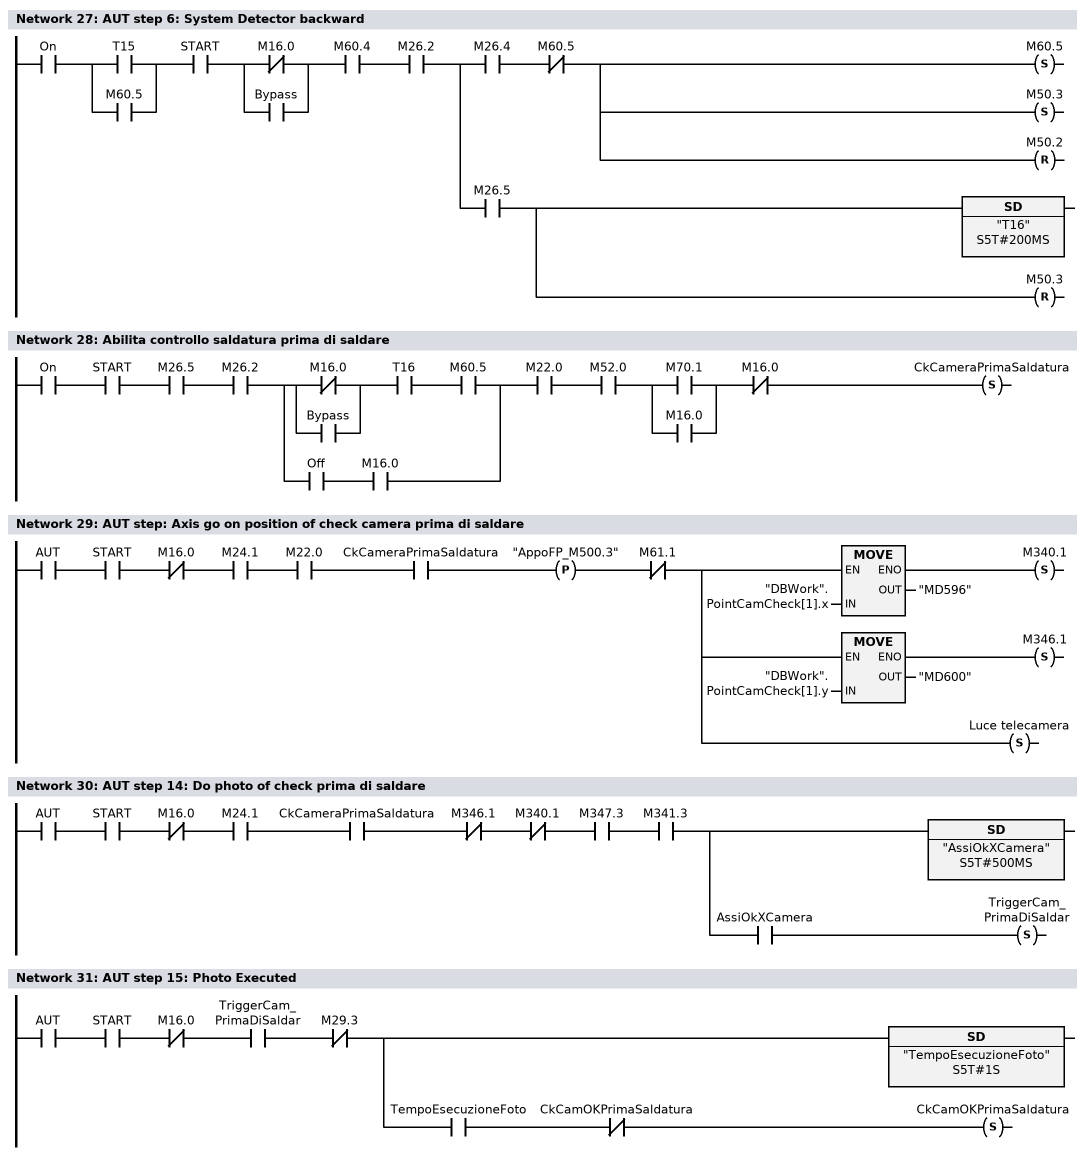
NETWORK
TITLE = AUT step 6: System Detector backward
//torno con il controllo in posizione iniziale
      A     "On";
      A(;
      O     "T15";
      O     "M60.5";
      );
      A     "START";
      A(;
      ON    "M16.0";
      O     "Bypass";
      );
      A     "M60.4";
      A     "M26.2";
      =     L 16.0;
      A     L 16.0;
      A     "M26.4";
      AN    "M60.5";
      S     "M60.5";
      S     "M50.3";
      R     "M50.2";
      A     L 16.0;
      A     "M26.5";
      L     S5T#200MS;
      SD    "T16";
      R     "M50.3";
NETWORK
TITLE = Abilita controllo saldatura prima di saldare
//System Detector in Pos initial and ready for detect Welding point
      A     "On";
      A     "START";
      A     "M26.5";
      A     "M26.2";
      A(;
      A(;
      ON    "M16.0";
      O     "Bypass";
      );
      A     "T16";
      A     "M60.5";
      O;
      A     "Off";
      A     "M16.0";
      );
      A     "M22.0";
      A     "M52.0";
      A(;
      O     "M70.1";
      O     "M16.0";
      );
      AN    "M16.0";
      S     "CkCameraPrimaSaldatura";
NETWORK
TITLE = AUT step: Axis go on position of check camera prima di saldare
      A     "AUT";
      A     "START";
      AN    "M16.0";
      A     "M24.1";
      A     "M22.0";
      A     "CkCameraPrimaSaldatura";
      FP    "AppoFP_M500.3";
      AN    "M61.1";
      =     L 16.0;
      A     L 16.0;
      JNB   _016;
      L     "DBWork".PointCamCheck[1].x;
      T     "MD596";
      SET;
      SAVE;
      CLR;
_016: A     BR;
      S     "M340.1";
      A     L 16.0;
      JNB   _017;
      L     "DBWork".PointCamCheck[1].y;
      T     "MD600";
      SET;
      SAVE;
      CLR;
_017: A     BR;
      S     "M346.1";
      A     L 16.0;
      BLD   102;
      S     "Luce telecamera";
NETWORK
TITLE = AUT step 14: Do photo of check prima di saldare
      A     "AUT";
      A     "START";
      AN    "M16.0";
      A     "M24.1";
      A     "CkCameraPrimaSaldatura";
      AN    "M346.1";
      AN    "M340.1";
      A     "M347.3";
      A     "M341.3";
      =     L 16.0;
      A     L 16.0;
      BLD   102;
      L     S5T#500MS;
      SD    "AssiOkXCamera";
      A     L 16.0;
      A     "AssiOkXCamera";
      S     "TriggerCam_PrimaDiSaldar";
NETWORK
TITLE = AUT step 15: Photo Executed
      A     "AUT";
      A     "START";
      AN    "M16.0";
      A     "TriggerCam_PrimaDiSaldar";
      AN    "M29.3";
      =     L 16.0;
      A     L 16.0;
      BLD   102;
      L     S5T#1S;
      SD    "TempoEsecuzioneFoto";
      A     L 16.0;
      A     "TempoEsecuzioneFoto";
      AN    "CkCamOKPrimaSaldatura";
      S     "CkCamOKPrimaSaldatura";
